LIN {X 0,Y 566.227,Z 211.515,A -85,B 0,C 180,E1 -2635.049,E2 -2635.049} C_VEL
LIN {X 0,Y 566.206,Z 211.459,A -85,B 0,C 180,E1 -2638.202,E2 -2638.202} C_VEL
LIN {X 0,Y 566.191,Z 211.454,A -85,B 0,C 180,E1 -2641.076,E2 -2641.076} C_VEL
LIN {X 0,Y 566.214,Z 211.456,A -85,B 0,C 180,E1 -2643.734,E2 -2643.734} C_VEL
LIN {X 0,Y 566.201,Z 211.452,A -85,B 0,C 180,E1 -2646.57,E2 -2646.57} C_VEL
LIN {X 0,Y 566.223,Z 211.456,A -85,B 0,C 180,E1 -2649.686,E2 -2649.686} C_VEL
LIN {X 0,Y 566.202,Z 211.451,A -85,B 0,C 180,E1 -2652.917,E2 -2652.917} C_VEL
LIN {X 0,Y 566.199,Z 211.455,A -85,B 0,C 180,E1 -2656.048,E2 -2656.048} C_VEL
LIN {X 0,Y 566.205,Z 211.454,A -85,B 0,C 180,E1 -2659.214,E2 -2659.214} C_VEL
LIN {X 0,Y 566.186,Z 211.462,A -85,B 0,C 180,E1 -2661.636,E2 -2661.636} C_VEL
LIN {X 0,Y 566.162,Z 211.455,A -85,B 0,C 180,E1 -2664.307,E2 -2664.307} C_VEL
LIN {X 0,Y 566.204,Z 211.45,A -85,B 0,C 180,E1 -2666.896,E2 -2666.896} C_VEL
LIN {X 0,Y 566.176,Z 211.464,A -85,B 0,C 180,E1 -2669.407,E2 -2669.407} C_VEL
LIN {X 0,Y 566.212,Z 211.45,A -85,B 0,C 180,E1 -2671.857,E2 -2671.857} C_VEL
LIN {X 0,Y 566.21,Z 211.448,A -85,B 0,C 180,E1 -2674.25,E2 -2674.25} C_VEL
LIN {X 0,Y 566.172,Z 211.456,A -85,B 0,C 180,E1 -2676.718,E2 -2676.718} C_VEL
LIN {X 0,Y 566.207,Z 211.45,A -85,B 0,C 180,E1 -2679.662,E2 -2679.662} C_VEL
LIN {X 0,Y 566.197,Z 211.45,A -85,B 0,C 180,E1 -2682.668,E2 -2682.668} C_VEL
LIN {X 0,Y 566.234,Z 211.449,A -85,B 0,C 180,E1 -2685.626,E2 -2685.626} C_VEL
LIN {X 0,Y 566.235,Z 211.449,A -85,B 0,C 180,E1 -2688.675,E2 -2688.675} C_VEL
LIN {X 0,Y 566.206,Z 211.451,A -85,B 0,C 180,E1 -2691.434,E2 -2691.434} C_VEL
LIN {X 0,Y 566.264,Z 211.444,A -85,B 0,C 180,E1 -2694.301,E2 -2694.301} C_VEL
LIN {X 0,Y 566.283,Z 211.439,A -85,B 0,C 180,E1 -2697.866,E2 -2697.866} C_VEL
LIN {X 0,Y 566.305,Z 211.441,A -85,B 0,C 180,E1 -2700.711,E2 -2700.711} C_VEL
LIN {X 0,Y 566.271,Z 211.45,A -85,B 0,C 180,E1 -2702.845,E2 -2702.845} C_VEL
LIN {X 0,Y 566.262,Z 211.443,A -85,B 0,C 180,E1 -2705.698,E2 -2705.698} C_VEL
LIN {X 0,Y 566.233,Z 211.454,A -85,B 0,C 180,E1 -2708.565,E2 -2708.565} C_VEL
LIN {X 0,Y 566.24,Z 211.444,A -85,B 0,C 180,E1 -2711.454,E2 -2711.454} C_VEL
LIN {X 0,Y 566.233,Z 211.457,A -85,B 0,C 180,E1 -2714.506,E2 -2714.506} C_VEL
LIN {X 0,Y 566.198,Z 211.45,A -85,B 0,C 180,E1 -2717.331,E2 -2717.331} C_VEL
LIN {X 0,Y 566.212,Z 211.454,A -85,B 0,C 180,E1 -2720.337,E2 -2720.337} C_VEL
LIN {X 0,Y 566.167,Z 211.455,A -85,B 0,C 180,E1 -2723.281,E2 -2723.281} C_VEL
LIN {X 0,Y 566.212,Z 211.451,A -85,B 0,C 180,E1 -2725.749,E2 -2725.749} C_VEL
LIN {X 0,Y 566.2,Z 211.448,A -85,B 0,C 180,E1 -2727.484,E2 -2727.484} C_VEL
LIN {X 0,Y 565.52,Z 211.54,A -85,B 0,C 180,E1 -2728.078,E2 -2728.078} C_VEL
LIN {X 0,Y 562.655,Z 211.899,A -85,B 0,C 180,E1 -2729.042,E2 -2729.042} C_VEL
LIN {X 0,Y 560.247,Z 212.2,A -85,B 0,C 180,E1 -2729.817,E2 -2729.817} C_VEL
LIN {X 0,Y 559.221,Z 212.327,A -85,B 0,C 180,E1 -2730.416,E2 -2730.416} C_VEL
LIN {X 0,Y 559.142,Z 212.333,A -85,B 0,C 180,E1 -2730.619,E2 -2730.619} C_VEL
LIN {X 0,Y 559.162,Z 212.329,A -85,B 0,C 180,E1 -2733.574,E2 -2733.574} C_VEL
LIN {X 0,Y 559.159,Z 212.333,A -85,B 0,C 180,E1 -2736.447,E2 -2736.447} C_VEL
LIN {X 0,Y 559.176,Z 212.326,A -85,B 0,C 180,E1 -2738.933,E2 -2738.933} C_VEL
LIN {X 0,Y 559.189,Z 212.329,A -85,B 0,C 180,E1 -2741.767,E2 -2741.767} C_VEL
LIN {X 0,Y 559.137,Z 212.33,A -85,B 0,C 180,E1 -2744.739,E2 -2744.739} C_VEL
LIN {X 0,Y 559.174,Z 212.327,A -85,B 0,C 180,E1 -2747.862,E2 -2747.862} C_VEL
LIN {X 0,Y 559.182,Z 212.33,A -85,B 0,C 180,E1 -2750.135,E2 -2750.135} C_VEL
LIN {X 0,Y 559.141,Z 212.331,A -85,B 0,C 180,E1 -2752.892,E2 -2752.892} C_VEL
LIN {X 0,Y 559.162,Z 212.331,A -85,B 0,C 180,E1 -2756.051,E2 -2756.051} C_VEL
LIN {X 0,Y 559.16,Z 212.33,A -85,B 0,C 180,E1 -2758.981,E2 -2758.981} C_VEL
LIN {X 0,Y 559.189,Z 212.326,A -85,B 0,C 180,E1 -2762.288,E2 -2762.288} C_VEL
LIN {X 0,Y 559.176,Z 212.328,A -85,B 0,C 180,E1 -2764.813,E2 -2764.813} C_VEL
LIN {X 0,Y 559.139,Z 212.335,A -85,B 0,C 180,E1 -2767.847,E2 -2767.847} C_VEL
LIN {X 0,Y 559.194,Z 212.325,A -85,B 0,C 180,E1 -2770.492,E2 -2770.492} C_VEL
LIN {X 0,Y 559.178,Z 212.335,A -85,B 0,C 180,E1 -2773.198,E2 -2773.198} C_VEL
LIN {X 0,Y 559.169,Z 212.328,A -85,B 0,C 180,E1 -2776.184,E2 -2776.184} C_VEL
LIN {X 0,Y 559.194,Z 212.333,A -85,B 0,C 180,E1 -2779.134,E2 -2779.134} C_VEL
LIN {X 0,Y 559.203,Z 212.324,A -85,B 0,C 180,E1 -2782.054,E2 -2782.054} C_VEL
LIN {X 0,Y 559.253,Z 212.325,A -85,B 0,C 180,E1 -2784.953,E2 -2784.953} C_VEL
LIN {X 0,Y 559.255,Z 212.318,A -85,B 0,C 180,E1 -2787.839,E2 -2787.839} C_VEL
LIN {X 0,Y 559.27,Z 212.322,A -85,B 0,C 180,E1 -2790.72,E2 -2790.72} C_VEL
LIN {X 0,Y 559.236,Z 212.328,A -85,B 0,C 180,E1 -2792.881,E2 -2792.881} C_VEL
LIN {X 0,Y 559.236,Z 212.32,A -85,B 0,C 180,E1 -2795.77,E2 -2795.77} C_VEL
LIN {X 0,Y 559.189,Z 212.333,A -85,B 0,C 180,E1 -2798.674,E2 -2798.674} C_VEL
LIN {X 0,Y 559.202,Z 212.325,A -85,B 0,C 180,E1 -2801.6,E2 -2801.6} C_VEL
LIN {X 0,Y 559.197,Z 212.333,A -85,B 0,C 180,E1 -2804.596,E2 -2804.596} C_VEL
LIN {X 0,Y 559.156,Z 212.33,A -85,B 0,C 180,E1 -2807.557,E2 -2807.557} C_VEL
LIN {X 0,Y 559.169,Z 212.329,A -85,B 0,C 180,E1 -2809.837,E2 -2809.837} C_VEL
LIN {X 0,Y 559.139,Z 212.335,A -85,B 0,C 180,E1 -2812.153,E2 -2812.153} C_VEL
LIN {X 0,Y 559.173,Z 212.328,A -85,B 0,C 180,E1 -2815.298,E2 -2815.298} C_VEL
LIN {X 0,Y 559.189,Z 212.326,A -85,B 0,C 180,E1 -2817.712,E2 -2817.712} C_VEL
LIN {X 0,Y 559.16,Z 212.33,A -85,B 0,C 180,E1 -2821.019,E2 -2821.019} C_VEL
LIN {X 0,Y 559.162,Z 212.331,A -85,B 0,C 180,E1 -2823.949,E2 -2823.949} C_VEL
LIN {X 0,Y 559.141,Z 212.331,A -85,B 0,C 180,E1 -2827.108,E2 -2827.108} C_VEL
LIN {X 0,Y 559.167,Z 212.333,A -85,B 0,C 180,E1 -2829.943,E2 -2829.943} C_VEL
LIN {X 0,Y 559.161,Z 212.324,A -85,B 0,C 180,E1 -2832.743,E2 -2832.743} C_VEL
LIN {X 0,Y 559.152,Z 212.333,A -85,B 0,C 180,E1 -2835.761,E2 -2835.761} C_VEL
LIN {X 0,Y 559.189,Z 212.329,A -85,B 0,C 180,E1 -2838.233,E2 -2838.233} C_VEL
LIN {X 0,Y 559.175,Z 212.327,A -85,B 0,C 180,E1 -2841.191,E2 -2841.191} C_VEL
LIN {X 0,Y 559.158,Z 212.336,A -85,B 0,C 180,E1 -2843.791,E2 -2843.791} C_VEL
LIN {X 0,Y 559.162,Z 212.329,A -85,B 0,C 180,E1 -2846.426,E2 -2846.426} C_VEL
LIN {X 0,Y 559.16,Z 212.329,A -85,B 0,C 180,E1 -2848.982,E2 -2848.982} C_VEL
LIN {X 0,Y 559.165,Z 212.334,A -85,B 0,C 180,E1 -2851.619,E2 -2851.619} C_VEL
LIN {X 0,Y 559.179,Z 212.332,A -85,B 0,C 180,E1 -2853.903,E2 -2853.903} C_VEL
LIN {X 0,Y 559.14,Z 212.331,A -85,B 0,C 180,E1 -2856.571,E2 -2856.571} C_VEL
LIN {X 0,Y 559.178,Z 212.331,A -85,B 0,C 180,E1 -2859.396,E2 -2859.396} C_VEL
LIN {X 0,Y 559.145,Z 212.336,A -85,B 0,C 180,E1 -2861.686,E2 -2861.686} C_VEL
LIN {X 0,Y 559.165,Z 212.331,A -85,B 0,C 180,E1 -2863.948,E2 -2863.948} C_VEL
LIN {X 0,Y 559.17,Z 212.328,A -85,B 0,C 180,E1 -2866.184,E2 -2866.184} C_VEL
LIN {X 0,Y 559.195,Z 212.326,A -85,B 0,C 180,E1 -2869.134,E2 -2869.134} C_VEL
LIN {X 0,Y 559.201,Z 212.322,A -85,B 0,C 180,E1 -2872.054,E2 -2872.054} C_VEL
LIN {X 0,Y 559.254,Z 212.321,A -85,B 0,C 180,E1 -2874.954,E2 -2874.954} C_VEL
LIN {X 0,Y 559.256,Z 212.315,A -85,B 0,C 180,E1 -2877.84,E2 -2877.84} C_VEL
LIN {X 0,Y 559.268,Z 212.312,A -85,B 0,C 180,E1 -2880.72,E2 -2880.72} C_VEL
LIN {X 0,Y 559.234,Z 212.323,A -85,B 0,C 180,E1 -2882.882,E2 -2882.882} C_VEL
LIN {X 0,Y 559.231,Z 212.32,A -85,B 0,C 180,E1 -2885.771,E2 -2885.771} C_VEL
LIN {X 0,Y 559.17,Z 212.328,A -85,B 0,C 180,E1 -2888.675,E2 -2888.675} C_VEL
LIN {X 0,Y 559.205,Z 212.322,A -85,B 0,C 180,E1 -2891.601,E2 -2891.601} C_VEL
LIN {X 0,Y 559.2,Z 212.328,A -85,B 0,C 180,E1 -2894.596,E2 -2894.596} C_VEL
LIN {X 0,Y 559.14,Z 212.327,A -85,B 0,C 180,E1 -2897.558,E2 -2897.558} C_VEL
LIN {X 0,Y 559.166,Z 212.324,A -85,B 0,C 180,E1 -2899.838,E2 -2899.838} C_VEL
LIN {X 0,Y 559.141,Z 212.331,A -85,B 0,C 180,E1 -2902.153,E2 -2902.153} C_VEL
LIN {X 0,Y 559.176,Z 212.325,A -85,B 0,C 180,E1 -2905.299,E2 -2905.299} C_VEL
LIN {X 0,Y 559.157,Z 212.325,A -85,B 0,C 180,E1 -2907.714,E2 -2907.714} C_VEL
LIN {X 0,Y 559.15,Z 212.333,A -85,B 0,C 180,E1 -2910.183,E2 -2910.183} C_VEL
LIN {X 0,Y 559.153,Z 212.333,A -85,B 0,C 180,E1 -2912.716,E2 -2912.716} C_VEL
LIN {X 0,Y 559.128,Z 212.331,A -85,B 0,C 180,E1 -2915.324,E2 -2915.324} C_VEL
LIN {X 0,Y 559.133,Z 212.335,A -85,B 0,C 180,E1 -2918.018,E2 -2918.018} C_VEL
LIN {X 0,Y 559.156,Z 212.332,A -85,B 0,C 180,E1 -2920.813,E2 -2920.813} C_VEL
LIN {X 0,Y 559.142,Z 212.332,A -85,B 0,C 180,E1 -2923.734,E2 -2923.734} C_VEL
LIN {X 0,Y 559.146,Z 212.332,A -85,B 0,C 180,E1 -2926.804,E2 -2926.804} C_VEL
LIN {X 0,Y 559.157,Z 212.325,A -85,B 0,C 180,E1 -2929.188,E2 -2929.188} C_VEL
LIN {X 0,Y 559.134,Z 212.338,A -85,B 0,C 180,E1 -2931.983,E2 -2931.983} C_VEL
LIN {X 0,Y 559.132,Z 212.332,A -85,B 0,C 180,E1 -2934.788,E2 -2934.788} C_VEL
LIN {X 0,Y 559.157,Z 212.33,A -85,B 0,C 180,E1 -2937.365,E2 -2937.365} C_VEL
LIN {X 0,Y 559.149,Z 212.337,A -85,B 0,C 180,E1 -2940.143,E2 -2940.143} C_VEL
LIN {X 0,Y 559.162,Z 212.332,A -85,B 0,C 180,E1 -2943.175,E2 -2943.175} C_VEL
LIN {X 0,Y 559.193,Z 212.546,A -85,B 0,C 180,E1 -2944.845,E2 -2944.845} C_VEL
LIN {X 0,Y 559.929,Z 217.985,A -85,B 0,C 180,E1 -2945.925,E2 -2945.925} C_VEL
LIN {X 0,Y 559.641,Z 232.53,A -85,B 0,C 180,E1 -2948.643,E2 -2948.643} C_VEL
LIN {X 0,Y 559.484,Z 246.129,A -85,B 0,C 180,E1 -2951.128,E2 -2951.128} C_VEL
LIN {X 0,Y 559.339,Z 260.753,A -85,B 0,C 180,E1 -2953.766,E2 -2953.766} C_VEL
LIN {X 0,Y 559.262,Z 272.268,A -85,B 0,C 180,E1 -2955.792,E2 -2955.792} C_VEL
LIN {X 0,Y 559.599,Z 274.63,A -85,B 0,C 180,E1 -2955.869,E2 -2955.869} C_VEL
LIN {X 0,Y 560.277,Z 280.09,A -85,B 0,C 180,E1 -2955.957,E2 -2955.957} C_VEL
LIN {X 0,Y 560.031,Z 378.524,A -85,B 0,C 180,E1 -2957.245,E2 -2957.245} C_VEL
LIN {X 0,Y 559.963,Z 388.812,A -85,B 0,C 180,E1 -2957.473,E2 -2957.473} C_VEL
LIN {X 0,Y 559.826,Z 399.596,A -85,B 0,C 180,E1 -2957.816,E2 -2957.816} C_VEL
LIN {X 0,Y 559.716,Z 412.055,A -85,B 0,C 180,E1 -2958.351,E2 -2958.351} C_VEL
LIN {X 0,Y 559.537,Z 424.284,A -85,B 0,C 180,E1 -2959.06,E2 -2959.06} C_VEL
LIN {X 0,Y 559.434,Z 433.031,A -85,B 0,C 180,E1 -2959.687,E2 -2959.687} C_VEL
LIN {X 0,Y 559.277,Z 441.533,A -85,B 0,C 180,E1 -2960.416,E2 -2960.416} C_VEL
LIN {X 0,Y 559.138,Z 448.723,A -85,B 0,C 180,E1 -2961.143,E2 -2961.143} C_VEL
LIN {X 0,Y 559.052,Z 456.27,A -85,B 0,C 180,E1 -2962.051,E2 -2962.051} C_VEL
LIN {X 0,Y 558.934,Z 462.674,A -85,B 0,C 180,E1 -2962.976,E2 -2962.976} C_VEL
LIN {X 0,Y 558.909,Z 467.794,A -85,B 0,C 180,E1 -2963.864,E2 -2963.864} C_VEL
LIN {X 0,Y 558.798,Z 472.891,A -85,B 0,C 180,E1 -2964.949,E2 -2964.949} C_VEL
LIN {X 0,Y 558.844,Z 476.848,A -85,B 0,C 180,E1 -2966.034,E2 -2966.034} C_VEL
LIN {X 0,Y 558.799,Z 479.771,A -85,B 0,C 180,E1 -2967.116,E2 -2967.116} C_VEL
LIN {X 0,Y 558.745,Z 482.196,A -85,B 0,C 180,E1 -2968.559,E2 -2968.559} C_VEL
LIN {X 0,Y 558.741,Z 482.78,A -85,B 0,C 180,E1 -2969.279,E2 -2969.279} C_VEL
LIN {X 0,Y 558.741,Z 482.78,A -85,B 0,C 180,E1 -2970.721,E2 -2970.721} C_VEL
LIN {X 0,Y 558.745,Z 482.196,A -85,B 0,C 180,E1 -2971.441,E2 -2971.441} C_VEL
LIN {X 0,Y 558.799,Z 479.771,A -85,B 0,C 180,E1 -2972.884,E2 -2972.884} C_VEL
LIN {X 0,Y 558.844,Z 476.848,A -85,B 0,C 180,E1 -2973.966,E2 -2973.966} C_VEL
LIN {X 0,Y 558.798,Z 472.891,A -85,B 0,C 180,E1 -2975.051,E2 -2975.051} C_VEL
LIN {X 0,Y 558.91,Z 467.794,A -85,B 0,C 180,E1 -2976.136,E2 -2976.136} C_VEL
LIN {X 0,Y 558.934,Z 462.674,A -85,B 0,C 180,E1 -2977.024,E2 -2977.024} C_VEL
LIN {X 0,Y 559.052,Z 456.27,A -85,B 0,C 180,E1 -2977.949,E2 -2977.949} C_VEL
LIN {X 0,Y 559.138,Z 448.723,A -85,B 0,C 180,E1 -2978.857,E2 -2978.857} C_VEL
LIN {X 0,Y 559.287,Z 439.616,A -85,B 0,C 180,E1 -2979.767,E2 -2979.767} C_VEL
LIN {X 0,Y 559.46,Z 428.158,A -85,B 0,C 180,E1 -2980.678,E2 -2980.678} C_VEL
LIN {X 0,Y 559.566,Z 419.19,A -85,B 0,C 180,E1 -2981.257,E2 -2981.257} C_VEL
LIN {X 0,Y 559.75,Z 408.68,A -85,B 0,C 180,E1 -2981.805,E2 -2981.805} C_VEL
LIN {X 0,Y 559.826,Z 399.596,A -85,B 0,C 180,E1 -2982.184,E2 -2982.184} C_VEL
LIN {X 0,Y 559.963,Z 388.812,A -85,B 0,C 180,E1 -2982.527,E2 -2982.527} C_VEL
LIN {X 0,Y 560.031,Z 378.524,A -85,B 0,C 180,E1 -2982.755,E2 -2982.755} C_VEL
LIN {X 0,Y 560.215,Z 278.301,A -85,B 0,C 180,E1 -2984.067,E2 -2984.067} C_VEL
LIN {X 0,Y 559.276,Z 272.599,A -85,B 0,C 180,E1 -2984.184,E2 -2984.184} C_VEL
LIN {X 0,Y 559.225,Z 271.167,A -85,B 0,C 180,E1 -2984.371,E2 -2984.371} C_VEL
LIN {X 0,Y 559.399,Z 254.896,A -85,B 0,C 180,E1 -2987.287,E2 -2987.287} C_VEL
LIN {X 0,Y 559.617,Z 238.81,A -85,B 0,C 180,E1 -2990.204,E2 -2990.204} C_VEL
LIN {X 0,Y 559.874,Z 222.392,A -85,B 0,C 180,E1 -2993.25,E2 -2993.25} C_VEL
LIN {X 0,Y 559.783,Z 215.926,A -85,B 0,C 180,E1 -2994.476,E2 -2994.476} C_VEL
LIN {X 0,Y 559.186,Z 212.411,A -85,B 0,C 180,E1 -2995.188,E2 -2995.188} C_VEL
LIN {X 0,Y 559.139,Z 212.339,A -85,B 0,C 180,E1 -2997.714,E2 -2997.714} C_VEL
LIN {X 0,Y 559.154,Z 212.338,A -85,B 0,C 180,E1 -3000.183,E2 -3000.183} C_VEL
LIN {X 0,Y 559.158,Z 212.329,A -85,B 0,C 180,E1 -3002.715,E2 -3002.715} C_VEL
LIN {X 0,Y 559.129,Z 212.334,A -85,B 0,C 180,E1 -3005.324,E2 -3005.324} C_VEL
LIN {X 0,Y 559.135,Z 212.338,A -85,B 0,C 180,E1 -3008.017,E2 -3008.017} C_VEL
LIN {X 0,Y 559.157,Z 212.325,A -85,B 0,C 180,E1 -3010.812,E2 -3010.812} C_VEL
LIN {X 0,Y 559.157,Z 212.338,A -85,B 0,C 180,E1 -3013.732,E2 -3013.732} C_VEL
LIN {X 0,Y 559.148,Z 212.33,A -85,B 0,C 180,E1 -3016.803,E2 -3016.803} C_VEL
LIN {X 0,Y 559.156,Z 212.332,A -85,B 0,C 180,E1 -3019.187,E2 -3019.187} C_VEL
LIN {X 0,Y 559.133,Z 212.335,A -85,B 0,C 180,E1 -3021.982,E2 -3021.982} C_VEL
LIN {X 0,Y 559.131,Z 212.331,A -85,B 0,C 180,E1 -3024.787,E2 -3024.787} C_VEL
LIN {X 0,Y 559.154,Z 212.335,A -85,B 0,C 180,E1 -3027.364,E2 -3027.364} C_VEL
LIN {X 0,Y 559.145,Z 212.33,A -85,B 0,C 180,E1 -3030.143,E2 -3030.143} C_VEL
LIN {X 0,Y 559.17,Z 212.33,A -85,B 0,C 180,E1 -3033.097,E2 -3033.097} C_VEL
LIN {X 0,Y 559.156,Z 212.335,A -85,B 0,C 180,E1 -3035.494,E2 -3035.494} C_VEL
LIN {X 0,Y 559.172,Z 212.328,A -85,B 0,C 180,E1 -3038.623,E2 -3038.623} C_VEL
LIN {X 0,Y 559.161,Z 212.33,A -85,B 0,C 180,E1 -3040.926,E2 -3040.926} C_VEL
LIN {X 0,Y 559.163,Z 212.327,A -85,B 0,C 180,E1 -3043.947,E2 -3043.947} C_VEL
LIN {X 0,Y 559.17,Z 212.327,A -85,B 0,C 180,E1 -3046.184,E2 -3046.184} C_VEL
LIN {X 0,Y 559.194,Z 212.326,A -85,B 0,C 180,E1 -3049.133,E2 -3049.133} C_VEL
LIN {X 0,Y 559.196,Z 212.321,A -85,B 0,C 180,E1 -3052.053,E2 -3052.053} C_VEL
LIN {X 0,Y 559.251,Z 212.326,A -85,B 0,C 180,E1 -3054.953,E2 -3054.953} C_VEL
LIN {X 0,Y 559.254,Z 212.315,A -85,B 0,C 180,E1 -3057.839,E2 -3057.839} C_VEL
LIN {X 0,Y 559.274,Z 212.316,A -85,B 0,C 180,E1 -3060.72,E2 -3060.72} C_VEL
LIN {X 0,Y 559.237,Z 212.326,A -85,B 0,C 180,E1 -3062.881,E2 -3062.881} C_VEL
LIN {X 0,Y 559.231,Z 212.319,A -85,B 0,C 180,E1 -3065.77,E2 -3065.77} C_VEL
LIN {X 0,Y 559.191,Z 212.328,A -85,B 0,C 180,E1 -3068.674,E2 -3068.674} C_VEL
LIN {X 0,Y 559.204,Z 212.32,A -85,B 0,C 180,E1 -3071.6,E2 -3071.6} C_VEL
LIN {X 0,Y 559.198,Z 212.332,A -85,B 0,C 180,E1 -3074.595,E2 -3074.595} C_VEL
LIN {X 0,Y 559.157,Z 212.326,A -85,B 0,C 180,E1 -3077.557,E2 -3077.557} C_VEL
LIN {X 0,Y 559.17,Z 212.324,A -85,B 0,C 180,E1 -3079.837,E2 -3079.837} C_VEL
LIN {X 0,Y 559.139,Z 212.336,A -85,B 0,C 180,E1 -3082.152,E2 -3082.152} C_VEL
LIN {X 0,Y 559.174,Z 212.325,A -85,B 0,C 180,E1 -3085.298,E2 -3085.298} C_VEL
LIN {X 0,Y 559.154,Z 212.326,A -85,B 0,C 180,E1 -3087.713,E2 -3087.713} C_VEL
LIN {X 0,Y 559.142,Z 212.333,A -85,B 0,C 180,E1 -3090.619,E2 -3090.619} C_VEL
LIN {X 0,Y 558.483,Z 212.415,A -85,B 0,C 180,E1 -3091.22,E2 -3091.22} C_VEL
LIN {X 0,Y 555.622,Z 212.777,A -85,B 0,C 180,E1 -3092.196,E2 -3092.196} C_VEL
LIN {X 0,Y 553.208,Z 213.072,A -85,B 0,C 180,E1 -3092.982,E2 -3092.982} C_VEL
LIN {X 0,Y 552.185,Z 213.198,A -85,B 0,C 180,E1 -3093.589,E2 -3093.589} C_VEL
LIN {X 0,Y 552.11,Z 213.209,A -85,B 0,C 180,E1 -3093.794,E2 -3093.794} C_VEL
LIN {X 0,Y 552.107,Z 213.208,A -85,B 0,C 180,E1 -3096.746,E2 -3096.746} C_VEL
LIN {X 0,Y 552.131,Z 213.206,A -85,B 0,C 180,E1 -3099.526,E2 -3099.526} C_VEL
LIN {X 0,Y 552.128,Z 213.207,A -85,B 0,C 180,E1 -3102.425,E2 -3102.425} C_VEL
LIN {X 0,Y 552.096,Z 213.212,A -85,B 0,C 180,E1 -3105.563,E2 -3105.563} C_VEL
LIN {X 0,Y 552.137,Z 213.197,A -85,B 0,C 180,E1 -3108.676,E2 -3108.676} C_VEL
LIN {X 0,Y 552.117,Z 213.209,A -85,B 0,C 180,E1 -3111.411,E2 -3111.411} C_VEL
LIN {X 0,Y 552.098,Z 213.207,A -85,B 0,C 180,E1 -3114.157,E2 -3114.157} C_VEL
LIN {X 0,Y 552.12,Z 213.204,A -85,B 0,C 180,E1 -3116.815,E2 -3116.815} C_VEL
LIN {X 0,Y 552.104,Z 213.214,A -85,B 0,C 180,E1 -3119.391,E2 -3119.391} C_VEL
LIN {X 0,Y 552.123,Z 213.21,A -85,B 0,C 180,E1 -3121.903,E2 -3121.903} C_VEL
LIN {X 0,Y 552.152,Z 213.202,A -85,B 0,C 180,E1 -3124.649,E2 -3124.649} C_VEL
LIN {X 0,Y 552.09,Z 213.218,A -85,B 0,C 180,E1 -3127.549,E2 -3127.549} C_VEL
LIN {X 0,Y 552.145,Z 213.203,A -85,B 0,C 180,E1 -3130.373,E2 -3130.373} C_VEL
LIN {X 0,Y 552.152,Z 213.207,A -85,B 0,C 180,E1 -3132.977,E2 -3132.977} C_VEL
LIN {X 0,Y 552.133,Z 213.206,A -85,B 0,C 180,E1 -3136.004,E2 -3136.004} C_VEL
LIN {X 0,Y 552.161,Z 213.208,A -85,B 0,C 180,E1 -3138.993,E2 -3138.993} C_VEL
LIN {X 0,Y 552.157,Z 213.203,A -85,B 0,C 180,E1 -3141.952,E2 -3141.952} C_VEL
LIN {X 0,Y 552.228,Z 213.199,A -85,B 0,C 180,E1 -3144.889,E2 -3144.889} C_VEL
LIN {X 0,Y 552.225,Z 213.194,A -85,B 0,C 180,E1 -3147.812,E2 -3147.812} C_VEL
LIN {X 0,Y 552.24,Z 213.198,A -85,B 0,C 180,E1 -3150.729,E2 -3150.729} C_VEL
LIN {X 0,Y 552.202,Z 213.204,A -85,B 0,C 180,E1 -3152.918,E2 -3152.918} C_VEL
LIN {X 0,Y 552.207,Z 213.196,A -85,B 0,C 180,E1 -3155.844,E2 -3155.844} C_VEL
LIN {X 0,Y 552.159,Z 213.21,A -85,B 0,C 180,E1 -3158.786,E2 -3158.786} C_VEL
LIN {X 0,Y 552.16,Z 213.202,A -85,B 0,C 180,E1 -3161.75,E2 -3161.75} C_VEL
LIN {X 0,Y 552.134,Z 213.213,A -85,B 0,C 180,E1 -3164.748,E2 -3164.748} C_VEL
LIN {X 0,Y 552.108,Z 213.208,A -85,B 0,C 180,E1 -3167.788,E2 -3167.788} C_VEL
LIN {X 0,Y 552.128,Z 213.208,A -85,B 0,C 180,E1 -3170.101,E2 -3170.101} C_VEL
LIN {X 0,Y 552.09,Z 213.218,A -85,B 0,C 180,E1 -3172.451,E2 -3172.451} C_VEL
LIN {X 0,Y 552.152,Z 213.202,A -85,B 0,C 180,E1 -3175.351,E2 -3175.351} C_VEL
LIN {X 0,Y 552.123,Z 213.21,A -85,B 0,C 180,E1 -3178.097,E2 -3178.097} C_VEL
LIN {X 0,Y 552.104,Z 213.214,A -85,B 0,C 180,E1 -3180.609,E2 -3180.609} C_VEL
LIN {X 0,Y 552.12,Z 213.204,A -85,B 0,C 180,E1 -3183.185,E2 -3183.185} C_VEL
LIN {X 0,Y 552.098,Z 213.207,A -85,B 0,C 180,E1 -3185.843,E2 -3185.843} C_VEL
LIN {X 0,Y 552.123,Z 213.205,A -85,B 0,C 180,E1 -3189.062,E2 -3189.062} C_VEL
LIN {X 0,Y 552.137,Z 213.198,A -85,B 0,C 180,E1 -3191.444,E2 -3191.444} C_VEL
LIN {X 0,Y 552.093,Z 213.211,A -85,B 0,C 180,E1 -3194.532,E2 -3194.532} C_VEL
LIN {X 0,Y 552.128,Z 213.207,A -85,B 0,C 180,E1 -3197.585,E2 -3197.585} C_VEL
LIN {X 0,Y 552.132,Z 213.206,A -85,B 0,C 180,E1 -3200.474,E2 -3200.474} C_VEL
LIN {X 0,Y 552.109,Z 213.208,A -85,B 0,C 180,E1 -3203.316,E2 -3203.316} C_VEL
LIN {X 0,Y 552.125,Z 213.211,A -85,B 0,C 180,E1 -3205.94,E2 -3205.94} C_VEL
LIN {X 0,Y 552.116,Z 213.207,A -85,B 0,C 180,E1 -3208.541,E2 -3208.541} C_VEL
LIN {X 0,Y 552.122,Z 213.208,A -85,B 0,C 180,E1 -3211.438,E2 -3211.438} C_VEL
LIN {X 0,Y 552.128,Z 213.204,A -85,B 0,C 180,E1 -3214.356,E2 -3214.356} C_VEL
LIN {X 0,Y 552.097,Z 213.208,A -85,B 0,C 180,E1 -3216.758,E2 -3216.758} C_VEL
LIN {X 0,Y 552.119,Z 213.207,A -85,B 0,C 180,E1 -3219.12,E2 -3219.12} C_VEL
LIN {X 0,Y 552.124,Z 213.206,A -85,B 0,C 180,E1 -3221.445,E2 -3221.445} C_VEL
LIN {X 0,Y 552.115,Z 213.212,A -85,B 0,C 180,E1 -3223.738,E2 -3223.738} C_VEL
LIN {X 0,Y 552.134,Z 213.205,A -85,B 0,C 180,E1 -3226.005,E2 -3226.005} C_VEL
LIN {X 0,Y 552.162,Z 213.2,A -85,B 0,C 180,E1 -3228.994,E2 -3228.994} C_VEL
LIN {X 0,Y 552.156,Z 213.2,A -85,B 0,C 180,E1 -3231.952,E2 -3231.952} C_VEL
LIN {X 0,Y 552.229,Z 213.195,A -85,B 0,C 180,E1 -3234.889,E2 -3234.889} C_VEL
LIN {X 0,Y 552.227,Z 213.19,A -85,B 0,C 180,E1 -3237.812,E2 -3237.812} C_VEL
LIN {X 0,Y 552.238,Z 213.187,A -85,B 0,C 180,E1 -3240.73,E2 -3240.73} C_VEL
LIN {X 0,Y 552.202,Z 213.199,A -85,B 0,C 180,E1 -3242.919,E2 -3242.919} C_VEL
LIN {X 0,Y 552.2,Z 213.195,A -85,B 0,C 180,E1 -3245.844,E2 -3245.844} C_VEL
LIN {X 0,Y 552.142,Z 213.205,A -85,B 0,C 180,E1 -3248.786,E2 -3248.786} C_VEL
LIN {X 0,Y 552.163,Z 213.198,A -85,B 0,C 180,E1 -3251.751,E2 -3251.751} C_VEL
LIN {X 0,Y 552.137,Z 213.21,A -85,B 0,C 180,E1 -3254.749,E2 -3254.749} C_VEL
LIN {X 0,Y 552.098,Z 213.203,A -85,B 0,C 180,E1 -3257.789,E2 -3257.789} C_VEL
LIN {X 0,Y 552.126,Z 213.201,A -85,B 0,C 180,E1 -3260.102,E2 -3260.102} C_VEL
LIN {X 0,Y 552.092,Z 213.213,A -85,B 0,C 180,E1 -3262.451,E2 -3262.451} C_VEL
LIN {X 0,Y 552.156,Z 213.199,A -85,B 0,C 180,E1 -3265.351,E2 -3265.351} C_VEL
LIN {X 0,Y 552.11,Z 213.205,A -85,B 0,C 180,E1 -3268.099,E2 -3268.099} C_VEL
LIN {X 0,Y 552.1,Z 213.217,A -85,B 0,C 180,E1 -3270.61,E2 -3270.61} C_VEL
LIN {X 0,Y 552.107,Z 213.205,A -85,B 0,C 180,E1 -3273.187,E2 -3273.187} C_VEL
LIN {X 0,Y 552.086,Z 213.21,A -85,B 0,C 180,E1 -3275.844,E2 -3275.844} C_VEL
LIN {X 0,Y 552.118,Z 213.211,A -85,B 0,C 180,E1 -3278.589,E2 -3278.589} C_VEL
LIN {X 0,Y 552.122,Z 213.205,A -85,B 0,C 180,E1 -3281.446,E2 -3281.446} C_VEL
LIN {X 0,Y 552.094,Z 213.214,A -85,B 0,C 180,E1 -3284.532,E2 -3284.532} C_VEL
LIN {X 0,Y 552.131,Z 213.205,A -85,B 0,C 180,E1 -3287.585,E2 -3287.585} C_VEL
LIN {X 0,Y 552.134,Z 213.208,A -85,B 0,C 180,E1 -3290.473,E2 -3290.473} C_VEL
LIN {X 0,Y 552.108,Z 213.207,A -85,B 0,C 180,E1 -3293.317,E2 -3293.317} C_VEL
LIN {X 0,Y 552.128,Z 213.211,A -85,B 0,C 180,E1 -3295.939,E2 -3295.939} C_VEL
LIN {X 0,Y 552.122,Z 213.209,A -85,B 0,C 180,E1 -3298.541,E2 -3298.541} C_VEL
LIN {X 0,Y 552.107,Z 213.212,A -85,B 0,C 180,E1 -3301.442,E2 -3301.442} C_VEL
LIN {X 0,Y 552.124,Z 213.213,A -85,B 0,C 180,E1 -3304.356,E2 -3304.356} C_VEL
LIN {X 0,Y 552.158,Z 213.415,A -85,B 0,C 180,E1 -3304.685,E2 -3304.685} C_VEL
LIN {X 0,Y 552.99,Z 218.935,A -85,B 0,C 180,E1 -3305.804,E2 -3305.804} C_VEL
LIN {X 0,Y 552.646,Z 234.49,A -85,B 0,C 180,E1 -3308.75,E2 -3308.75} C_VEL
LIN {X 0,Y 552.464,Z 248.087,A -85,B 0,C 180,E1 -3311.264,E2 -3311.264} C_VEL
LIN {X 0,Y 552.308,Z 262.71,A -85,B 0,C 180,E1 -3313.933,E2 -3313.933} C_VEL
LIN {X 0,Y 552.21,Z 272.104,A -85,B 0,C 180,E1 -3315.606,E2 -3315.606} C_VEL
LIN {X 0,Y 552.533,Z 274.407,A -85,B 0,C 180,E1 -3315.684,E2 -3315.684} C_VEL
LIN {X 0,Y 553.381,Z 280.27,A -85,B 0,C 180,E1 -3315.783,E2 -3315.783} C_VEL
LIN {X 0,Y 553.136,Z 377.099,A -85,B 0,C 180,E1 -3317.06,E2 -3317.06} C_VEL
LIN {X 0,Y 553.043,Z 387.872,A -85,B 0,C 180,E1 -3317.291,E2 -3317.291} C_VEL
LIN {X 0,Y 552.932,Z 396.977,A -85,B 0,C 180,E1 -3317.568,E2 -3317.568} C_VEL
LIN {X 0,Y 552.809,Z 406.337,A -85,B 0,C 180,E1 -3317.938,E2 -3317.938} C_VEL
LIN {X 0,Y 552.677,Z 416.63,A -85,B 0,C 180,E1 -3318.456,E2 -3318.456} C_VEL
LIN {X 0,Y 552.528,Z 425.443,A -85,B 0,C 180,E1 -3319.001,E2 -3319.001} C_VEL
LIN {X 0,Y 552.384,Z 434.149,A -85,B 0,C 180,E1 -3319.647,E2 -3319.647} C_VEL
LIN {X 0,Y 552.239,Z 441.521,A -85,B 0,C 180,E1 -3320.292,E2 -3320.292} C_VEL
LIN {X 0,Y 552.122,Z 448.714,A -85,B 0,C 180,E1 -3321.029,E2 -3321.029} C_VEL
LIN {X 0,Y 552.01,Z 454.891,A -85,B 0,C 180,E1 -3321.765,E2 -3321.765} C_VEL
LIN {X 0,Y 551.904,Z 461.399,A -85,B 0,C 180,E1 -3322.684,E2 -3322.684} C_VEL
LIN {X 0,Y 551.808,Z 467.088,A -85,B 0,C 180,E1 -3323.651,E2 -3323.651} C_VEL
LIN {X 0,Y 551.802,Z 471.338,A -85,B 0,C 180,E1 -3324.519,E2 -3324.519} C_VEL
LIN {X 0,Y 551.766,Z 475.632,A -85,B 0,C 180,E1 -3325.617,E2 -3325.617} C_VEL
LIN {X 0,Y 551.75,Z 477.975,A -85,B 0,C 180,E1 -3326.348,E2 -3326.348} C_VEL
LIN {X 0,Y 551.723,Z 479.764,A -85,B 0,C 180,E1 -3327.079,E2 -3327.079} C_VEL
LIN {X 0,Y 551.645,Z 482.191,A -85,B 0,C 180,E1 -3328.54,E2 -3328.54} C_VEL
LIN {X 0,Y 551.641,Z 482.775,A -85,B 0,C 180,E1 -3329.27,E2 -3329.27} C_VEL
LIN {X 0,Y 551.641,Z 482.775,A -85,B 0,C 180,E1 -3330.73,E2 -3330.73} C_VEL
LIN {X 0,Y 551.645,Z 482.191,A -85,B 0,C 180,E1 -3331.46,E2 -3331.46} C_VEL
LIN {X 0,Y 551.723,Z 479.764,A -85,B 0,C 180,E1 -3332.921,E2 -3332.921} C_VEL
LIN {X 0,Y 551.764,Z 476.84,A -85,B 0,C 180,E1 -3334.017,E2 -3334.017} C_VEL
LIN {X 0,Y 551.723,Z 472.882,A -85,B 0,C 180,E1 -3335.116,E2 -3335.116} C_VEL
LIN {X 0,Y 551.837,Z 468.388,A -85,B 0,C 180,E1 -3336.098,E2 -3336.098} C_VEL
LIN {X 0,Y 551.886,Z 462.549,A -85,B 0,C 180,E1 -3337.132,E2 -3337.132} C_VEL
LIN {X 0,Y 551.984,Z 456.261,A -85,B 0,C 180,E1 -3338.051,E2 -3338.051} C_VEL
LIN {X 0,Y 552.071,Z 450.334,A -85,B 0,C 180,E1 -3338.787,E2 -3338.787} C_VEL
LIN {X 0,Y 552.222,Z 443.434,A -85,B 0,C 180,E1 -3339.523,E2 -3339.523} C_VEL
LIN {X 0,Y 552.34,Z 435.28,A -85,B 0,C 180,E1 -3340.261,E2 -3340.261} C_VEL
LIN {X 0,Y 552.479,Z 426.792,A -85,B 0,C 180,E1 -3340.907,E2 -3340.907} C_VEL
LIN {X 0,Y 552.672,Z 417.641,A -85,B 0,C 180,E1 -3341.486,E2 -3341.486} C_VEL
LIN {X 0,Y 552.813,Z 408.352,A -85,B 0,C 180,E1 -3341.969,E2 -3341.969} C_VEL
LIN {X 0,Y 552.9,Z 399.554,A -85,B 0,C 180,E1 -3342.34,E2 -3342.34} C_VEL
LIN {X 0,Y 553.035,Z 389.622,A -85,B 0,C 180,E1 -3342.663,E2 -3342.663} C_VEL
LIN {X 0,Y 553.096,Z 379.762,A -85,B 0,C 180,E1 -3342.895,E2 -3342.895} C_VEL
LIN {X 0,Y 553.264,Z 355.152,A -85,B 0,C 180,E1 -3343.241,E2 -3343.241} C_VEL
LIN {X 0,Y 553.31,Z 278.875,A -85,B 0,C 180,E1 -3344.237,E2 -3344.237} C_VEL
LIN {X 0,Y 552.213,Z 272.296,A -85,B 0,C 180,E1 -3344.379,E2 -3344.379} C_VEL
LIN {X 0,Y 552.313,Z 260.622,A -85,B 0,C 180,E1 -3346.447,E2 -3346.447} C_VEL
LIN {X 0,Y 552.522,Z 245.997,A -85,B 0,C 180,E1 -3349.119,E2 -3349.119} C_VEL
LIN {X 0,Y 552.759,Z 231.34,A -85,B 0,C 180,E1 -3351.851,E2 -3351.851} C_VEL
LIN {X 0,Y 552.979,Z 218.96,A -85,B 0,C 180,E1 -3354.197,E2 -3354.197} C_VEL
LIN {X 0,Y 552.134,Z 213.236,A -85,B 0,C 180,E1 -3355.38,E2 -3355.38} C_VEL
LIN {X 0,Y 552.091,Z 213.217,A -85,B 0,C 180,E1 -3358.099,E2 -3358.099} C_VEL
LIN {X 0,Y 552.103,Z 213.211,A -85,B 0,C 180,E1 -3360.609,E2 -3360.609} C_VEL
LIN {X 0,Y 552.117,Z 213.206,A -85,B 0,C 180,E1 -3363.186,E2 -3363.186} C_VEL
LIN {X 0,Y 552.087,Z 213.215,A -85,B 0,C 180,E1 -3365.843,E2 -3365.843} C_VEL
LIN {X 0,Y 552.126,Z 213.205,A -85,B 0,C 180,E1 -3369.061,E2 -3369.061} C_VEL
LIN {X 0,Y 552.122,Z 213.205,A -85,B 0,C 180,E1 -3371.446,E2 -3371.446} C_VEL
LIN {X 0,Y 552.092,Z 213.209,A -85,B 0,C 180,E1 -3374.531,E2 -3374.531} C_VEL
LIN {X 0,Y 552.131,Z 213.212,A -85,B 0,C 180,E1 -3377.584,E2 -3377.584} C_VEL
LIN {X 0,Y 552.13,Z 213.202,A -85,B 0,C 180,E1 -3380.472,E2 -3380.472} C_VEL
LIN {X 0,Y 552.107,Z 213.213,A -85,B 0,C 180,E1 -3383.317,E2 -3383.317} C_VEL
LIN {X 0,Y 552.103,Z 213.207,A -85,B 0,C 180,E1 -3385.937,E2 -3385.937} C_VEL
LIN {X 0,Y 552.12,Z 213.205,A -85,B 0,C 180,E1 -3388.54,E2 -3388.54} C_VEL
LIN {X 0,Y 552.125,Z 213.21,A -85,B 0,C 180,E1 -3391.438,E2 -3391.438} C_VEL
LIN {X 0,Y 552.129,Z 213.201,A -85,B 0,C 180,E1 -3394.355,E2 -3394.355} C_VEL
LIN {X 0,Y 552.098,Z 213.21,A -85,B 0,C 180,E1 -3396.757,E2 -3396.757} C_VEL
LIN {X 0,Y 552.119,Z 213.213,A -85,B 0,C 180,E1 -3399.119,E2 -3399.119} C_VEL
LIN {X 0,Y 552.118,Z 213.206,A -85,B 0,C 180,E1 -3401.444,E2 -3401.444} C_VEL
LIN {X 0,Y 552.113,Z 213.206,A -85,B 0,C 180,E1 -3403.737,E2 -3403.737} C_VEL
LIN {X 0,Y 552.135,Z 213.203,A -85,B 0,C 180,E1 -3406.004,E2 -3406.004} C_VEL
LIN {X 0,Y 552.162,Z 213.204,A -85,B 0,C 180,E1 -3408.993,E2 -3408.993} C_VEL
LIN {X 0,Y 552.15,Z 213.198,A -85,B 0,C 180,E1 -3411.951,E2 -3411.951} C_VEL
LIN {X 0,Y 552.227,Z 213.201,A -85,B 0,C 180,E1 -3414.889,E2 -3414.889} C_VEL
LIN {X 0,Y 552.225,Z 213.19,A -85,B 0,C 180,E1 -3417.812,E2 -3417.812} C_VEL
LIN {X 0,Y 552.244,Z 213.191,A -85,B 0,C 180,E1 -3420.729,E2 -3420.729} C_VEL
LIN {X 0,Y 552.203,Z 213.201,A -85,B 0,C 180,E1 -3422.918,E2 -3422.918} C_VEL
LIN {X 0,Y 552.201,Z 213.195,A -85,B 0,C 180,E1 -3425.843,E2 -3425.843} C_VEL
LIN {X 0,Y 552.161,Z 213.201,A -85,B 0,C 180,E1 -3428.785,E2 -3428.785} C_VEL
LIN {X 0,Y 552.161,Z 213.197,A -85,B 0,C 180,E1 -3431.75,E2 -3431.75} C_VEL
LIN {X 0,Y 552.135,Z 213.209,A -85,B 0,C 180,E1 -3434.748,E2 -3434.748} C_VEL
LIN {X 0,Y 552.109,Z 213.205,A -85,B 0,C 180,E1 -3437.788,E2 -3437.788} C_VEL
LIN {X 0,Y 552.129,Z 213.203,A -85,B 0,C 180,E1 -3440.101,E2 -3440.101} C_VEL
LIN {X 0,Y 552.09,Z 213.217,A -85,B 0,C 180,E1 -3442.451,E2 -3442.451} C_VEL
LIN {X 0,Y 552.153,Z 213.2,A -85,B 0,C 180,E1 -3445.35,E2 -3445.35} C_VEL
LIN {X 0,Y 552.107,Z 213.209,A -85,B 0,C 180,E1 -3448.098,E2 -3448.098} C_VEL
LIN {X 0,Y 552.104,Z 213.211,A -85,B 0,C 180,E1 -3450.615,E2 -3450.615} C_VEL
LIN {X 0,Y 552.12,Z 213.204,A -85,B 0,C 180,E1 -3453.185,E2 -3453.185} C_VEL
LIN {X 0,Y 552.11,Z 213.209,A -85,B 0,C 180,E1 -3453.794,E2 -3453.794} C_VEL
LIN {X 0,Y 551.473,Z 213.293,A -85,B 0,C 180,E1 -3454.403,E2 -3454.403} C_VEL
LIN {X 0,Y 548.651,Z 213.645,A -85,B 0,C 180,E1 -3455.391,E2 -3455.391} C_VEL
LIN {X 0,Y 546.231,Z 213.947,A -85,B 0,C 180,E1 -3456.186,E2 -3456.186} C_VEL
LIN {X 0,Y 545.163,Z 214.073,A -85,B 0,C 180,E1 -3456.8,E2 -3456.8} C_VEL
LIN {X 0,Y 545.061,Z 214.085,A -85,B 0,C 180,E1 -3457.008,E2 -3457.008} C_VEL
LIN {X 0,Y 545.072,Z 214.087,A -85,B 0,C 180,E1 -3460.141,E2 -3460.141} C_VEL
LIN {X 0,Y 545.083,Z 214.082,A -85,B 0,C 180,E1 -3463.105,E2 -3463.105} C_VEL
LIN {X 0,Y 545.064,Z 214.082,A -85,B 0,C 180,E1 -3466.224,E2 -3466.224} C_VEL
LIN {X 0,Y 545.098,Z 214.073,A -85,B 0,C 180,E1 -3468.887,E2 -3468.887} C_VEL
LIN {X 0,Y 545.052,Z 214.095,A -85,B 0,C 180,E1 -3471.763,E2 -3471.763} C_VEL
LIN {X 0,Y 545.048,Z 214.082,A -85,B 0,C 180,E1 -3474.533,E2 -3474.533} C_VEL
LIN {X 0,Y 545.079,Z 214.084,A -85,B 0,C 180,E1 -3477.212,E2 -3477.212} C_VEL
LIN {X 0,Y 545.063,Z 214.086,A -85,B 0,C 180,E1 -3479.811,E2 -3479.811} C_VEL
LIN {X 0,Y 545.091,Z 214.082,A -85,B 0,C 180,E1 -3482.344,E2 -3482.344} C_VEL
LIN {X 0,Y 545.114,Z 214.08,A -85,B 0,C 180,E1 -3484.82,E2 -3484.82} C_VEL
LIN {X 0,Y 545.035,Z 214.095,A -85,B 0,C 180,E1 -3487.242,E2 -3487.242} C_VEL
LIN {X 0,Y 545.117,Z 214.079,A -85,B 0,C 180,E1 -3490.415,E2 -3490.415} C_VEL
LIN {X 0,Y 545.071,Z 214.091,A -85,B 0,C 180,E1 -3493.521,E2 -3493.521} C_VEL
LIN {X 0,Y 545.092,Z 214.084,A -85,B 0,C 180,E1 -3495.82,E2 -3495.82} C_VEL
LIN {X 0,Y 545.116,Z 214.083,A -85,B 0,C 180,E1 -3498.849,E2 -3498.849} C_VEL
LIN {X 0,Y 545.127,Z 214.079,A -85,B 0,C 180,E1 -3501.847,E2 -3501.847} C_VEL
LIN {X 0,Y 545.205,Z 214.074,A -85,B 0,C 180,E1 -3504.823,E2 -3504.823} C_VEL
LIN {X 0,Y 545.196,Z 214.07,A -85,B 0,C 180,E1 -3507.784,E2 -3507.784} C_VEL
LIN {X 0,Y 545.21,Z 214.074,A -85,B 0,C 180,E1 -3510.739,E2 -3510.739} C_VEL
LIN {X 0,Y 545.169,Z 214.08,A -85,B 0,C 180,E1 -3512.956,E2 -3512.956} C_VEL
LIN {X 0,Y 545.178,Z 214.072,A -85,B 0,C 180,E1 -3515.919,E2 -3515.919} C_VEL
LIN {X 0,Y 545.118,Z 214.087,A -85,B 0,C 180,E1 -3518.9,E2 -3518.9} C_VEL
LIN {X 0,Y 545.132,Z 214.078,A -85,B 0,C 180,E1 -3521.904,E2 -3521.904} C_VEL
LIN {X 0,Y 545.082,Z 214.089,A -85,B 0,C 180,E1 -3524.944,E2 -3524.944} C_VEL
LIN {X 0,Y 545.076,Z 214.086,A -85,B 0,C 180,E1 -3528.026,E2 -3528.026} C_VEL
LIN {X 0,Y 545.092,Z 214.088,A -85,B 0,C 180,E1 -3530.372,E2 -3530.372} C_VEL
LIN {X 0,Y 545.078,Z 214.084,A -85,B 0,C 180,E1 -3533.559,E2 -3533.559} C_VEL
LIN {X 0,Y 545.077,Z 214.086,A -85,B 0,C 180,E1 -3536.001,E2 -3536.001} C_VEL
LIN {X 0,Y 545.087,Z 214.081,A -85,B 0,C 180,E1 -3538.749,E2 -3538.749} C_VEL
LIN {X 0,Y 545.075,Z 214.085,A -85,B 0,C 180,E1 -3541.683,E2 -3541.683} C_VEL
LIN {X 0,Y 545.073,Z 214.084,A -85,B 0,C 180,E1 -3544.564,E2 -3544.564} C_VEL
LIN {X 0,Y 545.037,Z 214.088,A -85,B 0,C 180,E1 -3547.304,E2 -3547.304} C_VEL
LIN {X 0,Y 545.09,Z 214.085,A -85,B 0,C 180,E1 -3550.14,E2 -3550.14} C_VEL
LIN {X 0,Y 545.075,Z 214.076,A -85,B 0,C 180,E1 -3553.107,E2 -3553.107} C_VEL
LIN {X 0,Y 545.061,Z 214.092,A -85,B 0,C 180,E1 -3556.225,E2 -3556.225} C_VEL
LIN {X 0,Y 545.094,Z 214.078,A -85,B 0,C 180,E1 -3558.887,E2 -3558.887} C_VEL
LIN {X 0,Y 545.052,Z 214.092,A -85,B 0,C 180,E1 -3561.763,E2 -3561.763} C_VEL
LIN {X 0,Y 545.05,Z 214.084,A -85,B 0,C 180,E1 -3564.533,E2 -3564.533} C_VEL
LIN {X 0,Y 545.079,Z 214.082,A -85,B 0,C 180,E1 -3567.213,E2 -3567.213} C_VEL
LIN {X 0,Y 545.064,Z 214.093,A -85,B 0,C 180,E1 -3569.811,E2 -3569.811} C_VEL
LIN {X 0,Y 545.078,Z 214.078,A -85,B 0,C 180,E1 -3572.344,E2 -3572.344} C_VEL
LIN {X 0,Y 545.115,Z 214.077,A -85,B 0,C 180,E1 -3574.821,E2 -3574.821} C_VEL
LIN {X 0,Y 545.036,Z 214.091,A -85,B 0,C 180,E1 -3577.243,E2 -3577.243} C_VEL
LIN {X 0,Y 545.119,Z 214.071,A -85,B 0,C 180,E1 -3580.415,E2 -3580.415} C_VEL
LIN {X 0,Y 545.072,Z 214.09,A -85,B 0,C 180,E1 -3583.522,E2 -3583.522} C_VEL
LIN {X 0,Y 545.093,Z 214.085,A -85,B 0,C 180,E1 -3585.82,E2 -3585.82} C_VEL
LIN {X 0,Y 545.117,Z 214.076,A -85,B 0,C 180,E1 -3588.85,E2 -3588.85} C_VEL
LIN {X 0,Y 545.127,Z 214.077,A -85,B 0,C 180,E1 -3591.847,E2 -3591.847} C_VEL
LIN {X 0,Y 545.205,Z 214.069,A -85,B 0,C 180,E1 -3594.823,E2 -3594.823} C_VEL
LIN {X 0,Y 545.198,Z 214.065,A -85,B 0,C 180,E1 -3597.784,E2 -3597.784} C_VEL
LIN {X 0,Y 545.209,Z 214.062,A -85,B 0,C 180,E1 -3600.739,E2 -3600.739} C_VEL
LIN {X 0,Y 545.169,Z 214.076,A -85,B 0,C 180,E1 -3602.956,E2 -3602.956} C_VEL
LIN {X 0,Y 545.17,Z 214.071,A -85,B 0,C 180,E1 -3605.92,E2 -3605.92} C_VEL
LIN {X 0,Y 545.102,Z 214.082,A -85,B 0,C 180,E1 -3608.901,E2 -3608.901} C_VEL
LIN {X 0,Y 545.135,Z 214.073,A -85,B 0,C 180,E1 -3611.905,E2 -3611.905} C_VEL
LIN {X 0,Y 545.086,Z 214.089,A -85,B 0,C 180,E1 -3614.944,E2 -3614.944} C_VEL
LIN {X 0,Y 545.069,Z 214.078,A -85,B 0,C 180,E1 -3618.026,E2 -3618.026} C_VEL
LIN {X 0,Y 545.092,Z 214.08,A -85,B 0,C 180,E1 -3620.373,E2 -3620.373} C_VEL
LIN {X 0,Y 545.08,Z 214.082,A -85,B 0,C 180,E1 -3623.56,E2 -3623.56} C_VEL
LIN {X 0,Y 545.079,Z 214.08,A -85,B 0,C 180,E1 -3626.001,E2 -3626.001} C_VEL
LIN {X 0,Y 545.089,Z 214.088,A -85,B 0,C 180,E1 -3628.748,E2 -3628.748} C_VEL
LIN {X 0,Y 545.055,Z 214.086,A -85,B 0,C 180,E1 -3631.915,E2 -3631.915} C_VEL
LIN {X 0,Y 545.06,Z 214.09,A -85,B 0,C 180,E1 -3634.565,E2 -3634.565} C_VEL
LIN {X 0,Y 545.037,Z 214.088,A -85,B 0,C 180,E1 -3637.304,E2 -3637.304} C_VEL
LIN {X 0,Y 545.066,Z 214.088,A -85,B 0,C 180,E1 -3640.143,E2 -3640.143} C_VEL
LIN {X 0,Y 545.08,Z 214.083,A -85,B 0,C 180,E1 -3643.107,E2 -3643.107} C_VEL
LIN {X 0,Y 545.068,Z 214.093,A -85,B 0,C 180,E1 -3646.225,E2 -3646.225} C_VEL
LIN {X 0,Y 545.083,Z 214.078,A -85,B 0,C 180,E1 -3648.886,E2 -3648.886} C_VEL
LIN {X 0,Y 545.084,Z 214.083,A -85,B 0,C 180,E1 -3650.819,E2 -3650.819} C_VEL
LIN {X 0,Y 545.044,Z 214.089,A -85,B 0,C 180,E1 -3653.62,E2 -3653.62} C_VEL
LIN {X 0,Y 545.067,Z 214.089,A -85,B 0,C 180,E1 -3656.328,E2 -3656.328} C_VEL
LIN {X 0,Y 545.068,Z 214.086,A -85,B 0,C 180,E1 -3658.952,E2 -3658.952} C_VEL
LIN {X 0,Y 545.085,Z 214.087,A -85,B 0,C 180,E1 -3661.507,E2 -3661.507} C_VEL
LIN {X 0,Y 545.117,Z 214.186,A -85,B 0,C 180,E1 -3664.487,E2 -3664.487} C_VEL
LIN {X 0,Y 546.026,Z 219.885,A -85,B 0,C 180,E1 -3665.677,E2 -3665.677} C_VEL
LIN {X 0,Y 545.658,Z 235.412,A -85,B 0,C 180,E1 -3668.663,E2 -3668.663} C_VEL
LIN {X 0,Y 545.453,Z 249,A -85,B 0,C 180,E1 -3671.209,E2 -3671.209} C_VEL
LIN {X 0,Y 545.286,Z 263.623,A -85,B 0,C 180,E1 -3673.913,E2 -3673.913} C_VEL
LIN {X 0,Y 545.156,Z 272.133,A -85,B 0,C 180,E1 -3675.433,E2 -3675.433} C_VEL
LIN {X 0,Y 546.524,Z 281.026,A -85,B 0,C 180,E1 -3675.613,E2 -3675.613} C_VEL
LIN {X 0,Y 546.243,Z 376.907,A -85,B 0,C 180,E1 -3676.893,E2 -3676.893} C_VEL
LIN {X 0,Y 546.114,Z 386.805,A -85,B 0,C 180,E1 -3677.103,E2 -3677.103} C_VEL
LIN {X 0,Y 546.013,Z 396.785,A -85,B 0,C 180,E1 -3677.408,E2 -3677.408} C_VEL
LIN {X 0,Y 545.856,Z 406.144,A -85,B 0,C 180,E1 -3677.782,E2 -3677.782} C_VEL
LIN {X 0,Y 545.667,Z 416.454,A -85,B 0,C 180,E1 -3678.306,E2 -3678.306} C_VEL
LIN {X 0,Y 545.529,Z 425.291,A -85,B 0,C 180,E1 -3678.858,E2 -3678.858} C_VEL
LIN {X 0,Y 545.385,Z 434.023,A -85,B 0,C 180,E1 -3679.513,E2 -3679.513} C_VEL
LIN {X 0,Y 545.224,Z 441.421,A -85,B 0,C 180,E1 -3680.166,E2 -3680.166} C_VEL
LIN {X 0,Y 545.076,Z 448.642,A -85,B 0,C 180,E1 -3680.912,E2 -3680.912} C_VEL
LIN {X 0,Y 544.956,Z 454.844,A -85,B 0,C 180,E1 -3681.658,E2 -3681.658} C_VEL
LIN {X 0,Y 544.836,Z 461.381,A -85,B 0,C 180,E1 -3682.589,E2 -3682.589} C_VEL
LIN {X 0,Y 544.76,Z 466.255,A -85,B 0,C 180,E1 -3683.408,E2 -3683.408} C_VEL
LIN {X 0,Y 544.739,Z 471.328,A -85,B 0,C 180,E1 -3684.447,E2 -3684.447} C_VEL
LIN {X 0,Y 544.664,Z 475.624,A -85,B 0,C 180,E1 -3685.56,E2 -3685.56} C_VEL
LIN {X 0,Y 544.669,Z 477.972,A -85,B 0,C 180,E1 -3686.301,E2 -3686.301} C_VEL
LIN {X 0,Y 544.65,Z 479.758,A -85,B 0,C 180,E1 -3687.041,E2 -3687.041} C_VEL
LIN {X 0,Y 544.546,Z 482.183,A -85,B 0,C 180,E1 -3688.521,E2 -3688.521} C_VEL
LIN {X 0,Y 544.542,Z 482.766,A -85,B 0,C 180,E1 -3689.261,E2 -3689.261} C_VEL
LIN {X 0,Y 544.542,Z 482.766,A -85,B 0,C 180,E1 -3690.739,E2 -3690.739} C_VEL
LIN {X 0,Y 544.546,Z 482.183,A -85,B 0,C 180,E1 -3691.479,E2 -3691.479} C_VEL
LIN {X 0,Y 544.65,Z 479.758,A -85,B 0,C 180,E1 -3692.959,E2 -3692.959} C_VEL
LIN {X 0,Y 544.684,Z 476.832,A -85,B 0,C 180,E1 -3694.069,E2 -3694.069} C_VEL
LIN {X 0,Y 544.653,Z 472.872,A -85,B 0,C 180,E1 -3695.182,E2 -3695.182} C_VEL
LIN {X 0,Y 544.759,Z 468.63,A -85,B 0,C 180,E1 -3696.128,E2 -3696.128} C_VEL
LIN {X 0,Y 544.79,Z 463.688,A -85,B 0,C 180,E1 -3697.039,E2 -3697.039} C_VEL
LIN {X 0,Y 544.916,Z 457.596,A -85,B 0,C 180,E1 -3697.97,E2 -3697.97} C_VEL
LIN {X 0,Y 545,Z 451.896,A -85,B 0,C 180,E1 -3698.715,E2 -3698.715} C_VEL
LIN {X 0,Y 545.174,Z 443.34,A -85,B 0,C 180,E1 -3699.647,E2 -3699.647} C_VEL
LIN {X 0,Y 545.35,Z 435.158,A -85,B 0,C 180,E1 -3700.394,E2 -3700.394} C_VEL
LIN {X 0,Y 545.504,Z 426.643,A -85,B 0,C 180,E1 -3701.049,E2 -3701.049} C_VEL
LIN {X 0,Y 545.677,Z 418.185,A -85,B 0,C 180,E1 -3701.594,E2 -3701.594} C_VEL
LIN {X 0,Y 545.825,Z 409.167,A -85,B 0,C 180,E1 -3702.077,E2 -3702.077} C_VEL
LIN {X 0,Y 545.97,Z 399.361,A -85,B 0,C 180,E1 -3702.499,E2 -3702.499} C_VEL
LIN {X 0,Y 546.107,Z 389.429,A -85,B 0,C 180,E1 -3702.826,E2 -3702.826} C_VEL
LIN {X 0,Y 546.197,Z 379.57,A -85,B 0,C 180,E1 -3703.06,E2 -3703.06} C_VEL
LIN {X 0,Y 546.349,Z 354.96,A -85,B 0,C 180,E1 -3703.412,E2 -3703.412} C_VEL
LIN {X 0,Y 546.381,Z 279.325,A -85,B 0,C 180,E1 -3704.413,E2 -3704.413} C_VEL
LIN {X 0,Y 545.156,Z 272.129,A -85,B 0,C 180,E1 -3704.567,E2 -3704.567} C_VEL
LIN {X 0,Y 545.321,Z 258.403,A -85,B 0,C 180,E1 -3707.049,E2 -3707.049} C_VEL
LIN {X 0,Y 545.597,Z 243.09,A -85,B 0,C 180,E1 -3709.891,E2 -3709.891} C_VEL
LIN {X 0,Y 545.818,Z 227.171,A -85,B 0,C 180,E1 -3712.923,E2 -3712.923} C_VEL
LIN {X 0,Y 545.914,Z 218.869,A -85,B 0,C 180,E1 -3714.531,E2 -3714.531} C_VEL
LIN {X 0,Y 545.106,Z 214.11,A -85,B 0,C 180,E1 -3715.538,E2 -3715.538} C_VEL
LIN {X 0,Y 545.076,Z 214.086,A -85,B 0,C 180,E1 -3718.745,E2 -3718.745} C_VEL
LIN {X 0,Y 545.06,Z 214.092,A -85,B 0,C 180,E1 -3721.678,E2 -3721.678} C_VEL
LIN {X 0,Y 545.064,Z 214.085,A -85,B 0,C 180,E1 -3724.564,E2 -3724.564} C_VEL
LIN {X 0,Y 545.038,Z 214.089,A -85,B 0,C 180,E1 -3727.304,E2 -3727.304} C_VEL
LIN {X 0,Y 545.07,Z 214.083,A -85,B 0,C 180,E1 -3730.142,E2 -3730.142} C_VEL
LIN {X 0,Y 545.08,Z 214.084,A -85,B 0,C 180,E1 -3733.106,E2 -3733.106} C_VEL
LIN {X 0,Y 545.068,Z 214.086,A -85,B 0,C 180,E1 -3736.224,E2 -3736.224} C_VEL
LIN {X 0,Y 545.082,Z 214.082,A -85,B 0,C 180,E1 -3738.885,E2 -3738.885} C_VEL
LIN {X 0,Y 545.053,Z 214.092,A -85,B 0,C 180,E1 -3741.762,E2 -3741.762} C_VEL
LIN {X 0,Y 545.036,Z 214.086,A -85,B 0,C 180,E1 -3744.531,E2 -3744.531} C_VEL
LIN {X 0,Y 545.066,Z 214.086,A -85,B 0,C 180,E1 -3747.211,E2 -3747.211} C_VEL
LIN {X 0,Y 545.061,Z 214.088,A -85,B 0,C 180,E1 -3749.81,E2 -3749.81} C_VEL
LIN {X 0,Y 545.081,Z 214.078,A -85,B 0,C 180,E1 -3752.343,E2 -3752.343} C_VEL
LIN {X 0,Y 545.117,Z 214.077,A -85,B 0,C 180,E1 -3754.82,E2 -3754.82} C_VEL
LIN {X 0,Y 545.038,Z 214.096,A -85,B 0,C 180,E1 -3757.242,E2 -3757.242} C_VEL
LIN {X 0,Y 545.116,Z 214.074,A -85,B 0,C 180,E1 -3760.414,E2 -3760.414} C_VEL
LIN {X 0,Y 545.065,Z 214.086,A -85,B 0,C 180,E1 -3763.521,E2 -3763.521} C_VEL
LIN {X 0,Y 545.094,Z 214.081,A -85,B 0,C 180,E1 -3765.82,E2 -3765.82} C_VEL
LIN {X 0,Y 545.118,Z 214.082,A -85,B 0,C 180,E1 -3768.849,E2 -3768.849} C_VEL
LIN {X 0,Y 545.098,Z 214.076,A -85,B 0,C 180,E1 -3771.846,E2 -3771.846} C_VEL
LIN {X 0,Y 545.203,Z 214.075,A -85,B 0,C 180,E1 -3774.823,E2 -3774.823} C_VEL
LIN {X 0,Y 545.196,Z 214.066,A -85,B 0,C 180,E1 -3777.783,E2 -3777.783} C_VEL
LIN {X 0,Y 545.214,Z 214.066,A -85,B 0,C 180,E1 -3780.738,E2 -3780.738} C_VEL
LIN {X 0,Y 545.17,Z 214.077,A -85,B 0,C 180,E1 -3782.955,E2 -3782.955} C_VEL
LIN {X 0,Y 545.171,Z 214.071,A -85,B 0,C 180,E1 -3785.919,E2 -3785.919} C_VEL
LIN {X 0,Y 545.12,Z 214.075,A -85,B 0,C 180,E1 -3788.9,E2 -3788.9} C_VEL
LIN {X 0,Y 545.133,Z 214.073,A -85,B 0,C 180,E1 -3791.904,E2 -3791.904} C_VEL
LIN {X 0,Y 545.084,Z 214.085,A -85,B 0,C 180,E1 -3794.943,E2 -3794.943} C_VEL
LIN {X 0,Y 545.077,Z 214.083,A -85,B 0,C 180,E1 -3798.025,E2 -3798.025} C_VEL
LIN {X 0,Y 545.093,Z 214.084,A -85,B 0,C 180,E1 -3800.372,E2 -3800.372} C_VEL
LIN {X 0,Y 545.077,Z 214.083,A -85,B 0,C 180,E1 -3803.559,E2 -3803.559} C_VEL
LIN {X 0,Y 545.077,Z 214.086,A -85,B 0,C 180,E1 -3806,E2 -3806} C_VEL
LIN {X 0,Y 545.086,Z 214.082,A -85,B 0,C 180,E1 -3808.748,E2 -3808.748} C_VEL
LIN {X 0,Y 545.056,Z 214.088,A -85,B 0,C 180,E1 -3811.679,E2 -3811.679} C_VEL
LIN {X 0,Y 545.073,Z 214.083,A -85,B 0,C 180,E1 -3814.563,E2 -3814.563} C_VEL
LIN {X 0,Y 545.061,Z 214.085,A -85,B 0,C 180,E1 -3817.008,E2 -3817.008} C_VEL
LIN {X 0,Y 544.354,Z 214.178,A -85,B 0,C 180,E1 -3817.625,E2 -3817.625} C_VEL
LIN {X 0,Y 541.492,Z 214.533,A -85,B 0,C 180,E1 -3818.626,E2 -3818.626} C_VEL
LIN {X 0,Y 539.106,Z 214.83,A -85,B 0,C 180,E1 -3819.431,E2 -3819.431} C_VEL
LIN {X 0,Y 538.095,Z 214.957,A -85,B 0,C 180,E1 -3820.053,E2 -3820.053} C_VEL
LIN {X 0,Y 538.019,Z 214.961,A -85,B 0,C 180,E1 -3820.264,E2 -3820.264} C_VEL
LIN {X 0,Y 538.03,Z 214.961,A -85,B 0,C 180,E1 -3822.988,E2 -3822.988} C_VEL
LIN {X 0,Y 538.027,Z 214.962,A -85,B 0,C 180,E1 -3825.925,E2 -3825.925} C_VEL
LIN {X 0,Y 538.075,Z 214.949,A -85,B 0,C 180,E1 -3829.249,E2 -3829.249} C_VEL
LIN {X 0,Y 537.992,Z 214.97,A -85,B 0,C 180,E1 -3832.122,E2 -3832.122} C_VEL
LIN {X 0,Y 538.008,Z 214.959,A -85,B 0,C 180,E1 -3834.917,E2 -3834.917} C_VEL
LIN {X 0,Y 538.029,Z 214.968,A -85,B 0,C 180,E1 -3837.618,E2 -3837.618} C_VEL
LIN {X 0,Y 538.015,Z 214.959,A -85,B 0,C 180,E1 -3840.239,E2 -3840.239} C_VEL
LIN {X 0,Y 538.063,Z 214.958,A -85,B 0,C 180,E1 -3842.796,E2 -3842.796} C_VEL
LIN {X 0,Y 538.045,Z 214.966,A -85,B 0,C 180,E1 -3845.293,E2 -3845.293} C_VEL
LIN {X 0,Y 538.019,Z 214.963,A -85,B 0,C 180,E1 -3848.546,E2 -3848.546} C_VEL
LIN {X 0,Y 538.035,Z 214.964,A -85,B 0,C 180,E1 -3850.94,E2 -3850.94} C_VEL
LIN {X 0,Y 538.022,Z 214.971,A -85,B 0,C 180,E1 -3853.299,E2 -3853.299} C_VEL
LIN {X 0,Y 538.061,Z 214.963,A -85,B 0,C 180,E1 -3855.631,E2 -3855.631} C_VEL
LIN {X 0,Y 538.075,Z 214.959,A -85,B 0,C 180,E1 -3858.702,E2 -3858.702} C_VEL
LIN {X 0,Y 538.084,Z 214.958,A -85,B 0,C 180,E1 -3861.74,E2 -3861.74} C_VEL
LIN {X 0,Y 538.163,Z 214.95,A -85,B 0,C 180,E1 -3864.755,E2 -3864.755} C_VEL
LIN {X 0,Y 538.168,Z 214.946,A -85,B 0,C 180,E1 -3867.755,E2 -3867.755} C_VEL
LIN {X 0,Y 538.18,Z 214.949,A -85,B 0,C 180,E1 -3870.748,E2 -3870.748} C_VEL
LIN {X 0,Y 538.136,Z 214.957,A -85,B 0,C 180,E1 -3872.994,E2 -3872.994} C_VEL
LIN {X 0,Y 538.132,Z 214.95,A -85,B 0,C 180,E1 -3875.997,E2 -3875.997} C_VEL
LIN {X 0,Y 538.069,Z 214.964,A -85,B 0,C 180,E1 -3879.018,E2 -3879.018} C_VEL
LIN {X 0,Y 538.08,Z 214.957,A -85,B 0,C 180,E1 -3882.063,E2 -3882.063} C_VEL
LIN {X 0,Y 538.042,Z 214.964,A -85,B 0,C 180,E1 -3885.144,E2 -3885.144} C_VEL
LIN {X 0,Y 538.029,Z 214.966,A -85,B 0,C 180,E1 -3888.27,E2 -3888.27} C_VEL
LIN {X 0,Y 538.036,Z 214.969,A -85,B 0,C 180,E1 -3890.651,E2 -3890.651} C_VEL
LIN {X 0,Y 538.001,Z 214.967,A -85,B 0,C 180,E1 -3893.888,E2 -3893.888} C_VEL
LIN {X 0,Y 538.04,Z 214.968,A -85,B 0,C 180,E1 -3896.367,E2 -3896.367} C_VEL
LIN {X 0,Y 538.028,Z 214.957,A -85,B 0,C 180,E1 -3898.934,E2 -3898.934} C_VEL
LIN {X 0,Y 538.025,Z 214.965,A -85,B 0,C 180,E1 -3901.891,E2 -3901.891} C_VEL
LIN {X 0,Y 538.022,Z 214.961,A -85,B 0,C 180,E1 -3904.62,E2 -3904.62} C_VEL
LIN {X 0,Y 538.006,Z 214.964,A -85,B 0,C 180,E1 -3907.171,E2 -3907.171} C_VEL
LIN {X 0,Y 538.051,Z 214.961,A -85,B 0,C 180,E1 -3909.794,E2 -3909.794} C_VEL
LIN {X 0,Y 538.015,Z 214.956,A -85,B 0,C 180,E1 -3912.786,E2 -3912.786} C_VEL
LIN {X 0,Y 538.029,Z 214.959,A -85,B 0,C 180,E1 -3915.141,E2 -3915.141} C_VEL
LIN {X 0,Y 538.038,Z 214.963,A -85,B 0,C 180,E1 -3918.228,E2 -3918.228} C_VEL
LIN {X 0,Y 538.013,Z 214.963,A -85,B 0,C 180,E1 -3921.17,E2 -3921.17} C_VEL
LIN {X 0,Y 538.021,Z 214.965,A -85,B 0,C 180,E1 -3924.084,E2 -3924.084} C_VEL
LIN {X 0,Y 538.028,Z 214.959,A -85,B 0,C 180,E1 -3926.728,E2 -3926.728} C_VEL
LIN {X 0,Y 538.023,Z 214.967,A -85,B 0,C 180,E1 -3929.557,E2 -3929.557} C_VEL
LIN {X 0,Y 538.037,Z 214.96,A -85,B 0,C 180,E1 -3931.951,E2 -3931.951} C_VEL
LIN {X 0,Y 538.069,Z 214.955,A -85,B 0,C 180,E1 -3934.468,E2 -3934.468} C_VEL
LIN {X 0,Y 537.991,Z 214.972,A -85,B 0,C 180,E1 -3937.739,E2 -3937.739} C_VEL
LIN {X 0,Y 538.077,Z 214.95,A -85,B 0,C 180,E1 -3940.148,E2 -3940.148} C_VEL
LIN {X 0,Y 538.023,Z 214.964,A -85,B 0,C 180,E1 -3943.299,E2 -3943.299} C_VEL
LIN {X 0,Y 538.062,Z 214.963,A -85,B 0,C 180,E1 -3945.631,E2 -3945.631} C_VEL
LIN {X 0,Y 538.076,Z 214.952,A -85,B 0,C 180,E1 -3948.702,E2 -3948.702} C_VEL
LIN {X 0,Y 538.085,Z 214.955,A -85,B 0,C 180,E1 -3951.74,E2 -3951.74} C_VEL
LIN {X 0,Y 538.162,Z 214.946,A -85,B 0,C 180,E1 -3954.755,E2 -3954.755} C_VEL
LIN {X 0,Y 538.17,Z 214.941,A -85,B 0,C 180,E1 -3957.755,E2 -3957.755} C_VEL
LIN {X 0,Y 538.18,Z 214.937,A -85,B 0,C 180,E1 -3960.749,E2 -3960.749} C_VEL
LIN {X 0,Y 538.136,Z 214.952,A -85,B 0,C 180,E1 -3962.995,E2 -3962.995} C_VEL
LIN {X 0,Y 538.12,Z 214.949,A -85,B 0,C 180,E1 -3965.998,E2 -3965.998} C_VEL
LIN {X 0,Y 538.055,Z 214.957,A -85,B 0,C 180,E1 -3969.018,E2 -3969.018} C_VEL
LIN {X 0,Y 538.083,Z 214.951,A -85,B 0,C 180,E1 -3972.063,E2 -3972.063} C_VEL
LIN {X 0,Y 538.045,Z 214.962,A -85,B 0,C 180,E1 -3975.144,E2 -3975.144} C_VEL
LIN {X 0,Y 538.024,Z 214.957,A -85,B 0,C 180,E1 -3978.271,E2 -3978.271} C_VEL
LIN {X 0,Y 538.037,Z 214.962,A -85,B 0,C 180,E1 -3980.652,E2 -3980.652} C_VEL
LIN {X 0,Y 538.003,Z 214.964,A -85,B 0,C 180,E1 -3983.889,E2 -3983.889} C_VEL
LIN {X 0,Y 538.042,Z 214.96,A -85,B 0,C 180,E1 -3986.367,E2 -3986.367} C_VEL
LIN {X 0,Y 538.03,Z 214.965,A -85,B 0,C 180,E1 -3988.934,E2 -3988.934} C_VEL
LIN {X 0,Y 538.01,Z 214.964,A -85,B 0,C 180,E1 -3991.887,E2 -3991.887} C_VEL
LIN {X 0,Y 538.01,Z 214.968,A -85,B 0,C 180,E1 -3994.618,E2 -3994.618} C_VEL
LIN {X 0,Y 538.005,Z 214.965,A -85,B 0,C 180,E1 -3997.17,E2 -3997.17} C_VEL
LIN {X 0,Y 538.023,Z 214.961,A -85,B 0,C 180,E1 -3999.797,E2 -3999.797} C_VEL
LIN {X 0,Y 538.02,Z 214.965,A -85,B 0,C 180,E1 -4002.786,E2 -4002.786} C_VEL
LIN {X 0,Y 538.008,Z 214.963,A -85,B 0,C 180,E1 -4005.138,E2 -4005.138} C_VEL
LIN {X 0,Y 538.032,Z 214.965,A -85,B 0,C 180,E1 -4008.227,E2 -4008.227} C_VEL
LIN {X 0,Y 538.016,Z 214.962,A -85,B 0,C 180,E1 -4011.17,E2 -4011.17} C_VEL
LIN {X 0,Y 537.996,Z 214.969,A -85,B 0,C 180,E1 -4014.089,E2 -4014.089} C_VEL
LIN {X 0,Y 538.033,Z 214.961,A -85,B 0,C 180,E1 -4016.728,E2 -4016.728} C_VEL
LIN {X 0,Y 538.029,Z 214.966,A -85,B 0,C 180,E1 -4019.557,E2 -4019.557} C_VEL
LIN {X 0,Y 538.032,Z 214.966,A -85,B 0,C 180,E1 -4022.654,E2 -4022.654} C_VEL
LIN {X 0,Y 538.071,Z 215.154,A -85,B 0,C 180,E1 -4024.358,E2 -4024.358} C_VEL
LIN {X 0,Y 539.076,Z 221.41,A -85,B 0,C 180,E1 -4025.663,E2 -4025.663} C_VEL
LIN {X 0,Y 538.712,Z 238.409,A -85,B 0,C 180,E1 -4028.976,E2 -4028.976} C_VEL
LIN {X 0,Y 538.452,Z 253.049,A -85,B 0,C 180,E1 -4031.745,E2 -4031.745} C_VEL
LIN {X 0,Y 538.146,Z 269.679,A -85,B 0,C 180,E1 -4034.859,E2 -4034.859} C_VEL
LIN {X 0,Y 538.137,Z 271.942,A -85,B 0,C 180,E1 -4035.24,E2 -4035.24} C_VEL
LIN {X 0,Y 539.663,Z 281.867,A -85,B 0,C 180,E1 -4035.44,E2 -4035.44} C_VEL
LIN {X 0,Y 539.33,Z 376.714,A -85,B 0,C 180,E1 -4036.722,E2 -4036.722} C_VEL
LIN {X 0,Y 539.185,Z 387.487,A -85,B 0,C 180,E1 -4036.958,E2 -4036.958} C_VEL
LIN {X 0,Y 539.072,Z 396.592,A -85,B 0,C 180,E1 -4037.243,E2 -4037.243} C_VEL
LIN {X 0,Y 538.906,Z 405.951,A -85,B 0,C 180,E1 -4037.622,E2 -4037.622} C_VEL
LIN {X 0,Y 538.73,Z 415.592,A -85,B 0,C 180,E1 -4038.114,E2 -4038.114} C_VEL
LIN {X 0,Y 538.535,Z 425.097,A -85,B 0,C 180,E1 -4038.711,E2 -4038.711} C_VEL
LIN {X 0,Y 538.368,Z 433.83,A -85,B 0,C 180,E1 -4039.374,E2 -4039.374} C_VEL
LIN {X 0,Y 538.187,Z 441.227,A -85,B 0,C 180,E1 -4040.036,E2 -4040.036} C_VEL
LIN {X 0,Y 538.014,Z 448.448,A -85,B 0,C 180,E1 -4040.792,E2 -4040.792} C_VEL
LIN {X 0,Y 537.906,Z 454.651,A -85,B 0,C 180,E1 -4041.548,E2 -4041.548} C_VEL
LIN {X 0,Y 537.754,Z 461.187,A -85,B 0,C 180,E1 -4042.49,E2 -4042.49} C_VEL
LIN {X 0,Y 537.673,Z 466.577,A -85,B 0,C 180,E1 -4043.419,E2 -4043.419} C_VEL
LIN {X 0,Y 537.653,Z 471.176,A -85,B 0,C 180,E1 -4044.374,E2 -4044.374} C_VEL
LIN {X 0,Y 537.56,Z 475.494,A -85,B 0,C 180,E1 -4045.501,E2 -4045.501} C_VEL
LIN {X 0,Y 537.591,Z 477.858,A -85,B 0,C 180,E1 -4046.252,E2 -4046.252} C_VEL
LIN {X 0,Y 537.551,Z 479.652,A -85,B 0,C 180,E1 -4047.002,E2 -4047.002} C_VEL
LIN {X 0,Y 537.451,Z 482.089,A -85,B 0,C 180,E1 -4048.501,E2 -4048.501} C_VEL
LIN {X 0,Y 537.442,Z 482.676,A -85,B 0,C 180,E1 -4049.251,E2 -4049.251} C_VEL
LIN {X 0,Y 537.442,Z 482.676,A -85,B 0,C 180,E1 -4050.749,E2 -4050.749} C_VEL
LIN {X 0,Y 537.451,Z 482.089,A -85,B 0,C 180,E1 -4051.499,E2 -4051.499} C_VEL
LIN {X 0,Y 537.551,Z 479.652,A -85,B 0,C 180,E1 -4052.998,E2 -4052.998} C_VEL
LIN {X 0,Y 537.604,Z 476.711,A -85,B 0,C 180,E1 -4054.123,E2 -4054.123} C_VEL
LIN {X 0,Y 537.586,Z 472.727,A -85,B 0,C 180,E1 -4055.251,E2 -4055.251} C_VEL
LIN {X 0,Y 537.63,Z 467.911,A -85,B 0,C 180,E1 -4056.318,E2 -4056.318} C_VEL
LIN {X 0,Y 537.754,Z 462.343,A -85,B 0,C 180,E1 -4057.321,E2 -4057.321} C_VEL
LIN {X 0,Y 537.873,Z 456.027,A -85,B 0,C 180,E1 -4058.264,E2 -4058.264} C_VEL
LIN {X 0,Y 537.98,Z 450.075,A -85,B 0,C 180,E1 -4059.019,E2 -4059.019} C_VEL
LIN {X 0,Y 538.132,Z 443.146,A -85,B 0,C 180,E1 -4059.775,E2 -4059.775} C_VEL
LIN {X 0,Y 538.305,Z 436.1,A -85,B 0,C 180,E1 -4060.437,E2 -4060.437} C_VEL
LIN {X 0,Y 538.482,Z 427.802,A -85,B 0,C 180,E1 -4061.099,E2 -4061.099} C_VEL
LIN {X 0,Y 538.694,Z 418.055,A -85,B 0,C 180,E1 -4061.743,E2 -4061.743} C_VEL
LIN {X 0,Y 538.881,Z 407.966,A -85,B 0,C 180,E1 -4062.283,E2 -4062.283} C_VEL
LIN {X 0,Y 539.021,Z 399.168,A -85,B 0,C 180,E1 -4062.663,E2 -4062.663} C_VEL
LIN {X 0,Y 539.164,Z 389.236,A -85,B 0,C 180,E1 -4062.994,E2 -4062.994} C_VEL
LIN {X 0,Y 539.3,Z 379.378,A -85,B 0,C 180,E1 -4063.23,E2 -4063.23} C_VEL
LIN {X 0,Y 539.453,Z 354.767,A -85,B 0,C 180,E1 -4063.586,E2 -4063.586} C_VEL
LIN {X 0,Y 539.608,Z 280.704,A -85,B 0,C 180,E1 -4064.577,E2 -4064.577} C_VEL
LIN {X 0,Y 538.125,Z 271.938,A -85,B 0,C 180,E1 -4064.761,E2 -4064.761} C_VEL
LIN {X 0,Y 538.157,Z 268.69,A -85,B 0,C 180,E1 -4065.334,E2 -4065.334} C_VEL
LIN {X 0,Y 538.422,Z 252.003,A -85,B 0,C 180,E1 -4068.453,E2 -4068.453} C_VEL
LIN {X 0,Y 538.678,Z 238.409,A -85,B 0,C 180,E1 -4071.026,E2 -4071.026} C_VEL
LIN {X 0,Y 539.032,Z 222.507,A -85,B 0,C 180,E1 -4074.122,E2 -4074.122} C_VEL
LIN {X 0,Y 538.557,Z 217.715,A -85,B 0,C 180,E1 -4075.095,E2 -4075.095} C_VEL
LIN {X 0,Y 538.05,Z 214.989,A -85,B 0,C 180,E1 -4075.709,E2 -4075.709} C_VEL
LIN {X 0,Y 538.023,Z 214.968,A -85,B 0,C 180,E1 -4078.051,E2 -4078.051} C_VEL
LIN {X 0,Y 538.023,Z 214.965,A -85,B 0,C 180,E1 -4080.627,E2 -4080.627} C_VEL
LIN {X 0,Y 538.048,Z 214.96,A -85,B 0,C 180,E1 -4083.282,E2 -4083.282} C_VEL
LIN {X 0,Y 537.996,Z 214.97,A -85,B 0,C 180,E1 -4086.004,E2 -4086.004} C_VEL
LIN {X 0,Y 538.016,Z 214.962,A -85,B 0,C 180,E1 -4088.83,E2 -4088.83} C_VEL
LIN {X 0,Y 538.032,Z 214.965,A -85,B 0,C 180,E1 -4091.773,E2 -4091.773} C_VEL
LIN {X 0,Y 538.008,Z 214.963,A -85,B 0,C 180,E1 -4094.862,E2 -4094.862} C_VEL
LIN {X 0,Y 538.02,Z 214.965,A -85,B 0,C 180,E1 -4097.214,E2 -4097.214} C_VEL
LIN {X 0,Y 538.023,Z 214.961,A -85,B 0,C 180,E1 -4100.203,E2 -4100.203} C_VEL
LIN {X 0,Y 538.025,Z 214.964,A -85,B 0,C 180,E1 -4103.067,E2 -4103.067} C_VEL
LIN {X 0,Y 538.011,Z 214.963,A -85,B 0,C 180,E1 -4105.826,E2 -4105.826} C_VEL
LIN {X 0,Y 538.009,Z 214.963,A -85,B 0,C 180,E1 -4108.498,E2 -4108.498} C_VEL
LIN {X 0,Y 538.043,Z 214.964,A -85,B 0,C 180,E1 -4111.099,E2 -4111.099} C_VEL
LIN {X 0,Y 538.042,Z 214.96,A -85,B 0,C 180,E1 -4113.633,E2 -4113.633} C_VEL
LIN {X 0,Y 538.007,Z 214.963,A -85,B 0,C 180,E1 -4116.122,E2 -4116.122} C_VEL
LIN {X 0,Y 538.037,Z 214.962,A -85,B 0,C 180,E1 -4119.348,E2 -4119.348} C_VEL
LIN {X 0,Y 538.036,Z 214.955,A -85,B 0,C 180,E1 -4122.467,E2 -4122.467} C_VEL
LIN {X 0,Y 538.064,Z 214.958,A -85,B 0,C 180,E1 -4125.63,E2 -4125.63} C_VEL
LIN {X 0,Y 538.077,Z 214.956,A -85,B 0,C 180,E1 -4128.701,E2 -4128.701} C_VEL
LIN {X 0,Y 538.061,Z 214.953,A -85,B 0,C 180,E1 -4131.739,E2 -4131.739} C_VEL
LIN {X 0,Y 538.16,Z 214.951,A -85,B 0,C 180,E1 -4134.755,E2 -4134.755} C_VEL
LIN {X 0,Y 538.168,Z 214.941,A -85,B 0,C 180,E1 -4137.754,E2 -4137.754} C_VEL
LIN {X 0,Y 538.183,Z 214.941,A -85,B 0,C 180,E1 -4140.748,E2 -4140.748} C_VEL
LIN {X 0,Y 538.136,Z 214.952,A -85,B 0,C 180,E1 -4142.994,E2 -4142.994} C_VEL
LIN {X 0,Y 538.121,Z 214.95,A -85,B 0,C 180,E1 -4145.997,E2 -4145.997} C_VEL
LIN {X 0,Y 538.07,Z 214.951,A -85,B 0,C 180,E1 -4149.017,E2 -4149.017} C_VEL
LIN {X 0,Y 538.082,Z 214.953,A -85,B 0,C 180,E1 -4152.062,E2 -4152.062} C_VEL
LIN {X 0,Y 538.044,Z 214.96,A -85,B 0,C 180,E1 -4155.143,E2 -4155.143} C_VEL
LIN {X 0,Y 538.03,Z 214.964,A -85,B 0,C 180,E1 -4158.27,E2 -4158.27} C_VEL
LIN {X 0,Y 538.037,Z 214.963,A -85,B 0,C 180,E1 -4160.651,E2 -4160.651} C_VEL
LIN {X 0,Y 538,Z 214.968,A -85,B 0,C 180,E1 -4163.888,E2 -4163.888} C_VEL
LIN {X 0,Y 538.039,Z 214.961,A -85,B 0,C 180,E1 -4166.366,E2 -4166.366} C_VEL
LIN {X 0,Y 538.028,Z 214.96,A -85,B 0,C 180,E1 -4168.933,E2 -4168.933} C_VEL
LIN {X 0,Y 538.012,Z 214.968,A -85,B 0,C 180,E1 -4171.888,E2 -4171.888} C_VEL
LIN {X 0,Y 538.023,Z 214.96,A -85,B 0,C 180,E1 -4174.62,E2 -4174.62} C_VEL
LIN {X 0,Y 538.004,Z 214.964,A -85,B 0,C 180,E1 -4177.17,E2 -4177.17} C_VEL
LIN {X 0,Y 538.019,Z 214.961,A -85,B 0,C 180,E1 -4180.264,E2 -4180.264} C_VEL
LIN {X 0,Y 537.369,Z 215.041,A -85,B 0,C 180,E1 -4180.889,E2 -4180.889} C_VEL
LIN {X 0,Y 534.519,Z 215.403,A -85,B 0,C 180,E1 -4181.904,E2 -4181.904} C_VEL
LIN {X 0,Y 532.096,Z 215.707,A -85,B 0,C 180,E1 -4182.721,E2 -4182.721} C_VEL
LIN {X 0,Y 531.048,Z 215.835,A -85,B 0,C 180,E1 -4183.352,E2 -4183.352} C_VEL
LIN {X 0,Y 530.96,Z 215.844,A -85,B 0,C 180,E1 -4183.566,E2 -4183.566} C_VEL
LIN {X 0,Y 530.961,Z 215.834,A -85,B 0,C 180,E1 -4186.505,E2 -4186.505} C_VEL
LIN {X 0,Y 531.023,Z 215.831,A -85,B 0,C 180,E1 -4189.571,E2 -4189.571} C_VEL
LIN {X 0,Y 530.966,Z 215.841,A -85,B 0,C 180,E1 -4192.576,E2 -4192.576} C_VEL
LIN {X 0,Y 530.992,Z 215.836,A -85,B 0,C 180,E1 -4195.311,E2 -4195.311} C_VEL
LIN {X 0,Y 530.98,Z 215.843,A -85,B 0,C 180,E1 -4198.033,E2 -4198.033} C_VEL
LIN {X 0,Y 530.986,Z 215.833,A -85,B 0,C 180,E1 -4200.874,E2 -4200.874} C_VEL
LIN {X 0,Y 531.003,Z 215.842,A -85,B 0,C 180,E1 -4203.256,E2 -4203.256} C_VEL
LIN {X 0,Y 530.982,Z 215.843,A -85,B 0,C 180,E1 -4205.96,E2 -4205.96} C_VEL
LIN {X 0,Y 530.997,Z 215.842,A -85,B 0,C 180,E1 -4209.062,E2 -4209.062} C_VEL
LIN {X 0,Y 531.013,Z 215.837,A -85,B 0,C 180,E1 -4212.278,E2 -4212.278} C_VEL
LIN {X 0,Y 531.037,Z 215.84,A -85,B 0,C 180,E1 -4215.436,E2 -4215.436} C_VEL
LIN {X 0,Y 531.034,Z 215.835,A -85,B 0,C 180,E1 -4218.55,E2 -4218.55} C_VEL
LIN {X 0,Y 531.054,Z 215.835,A -85,B 0,C 180,E1 -4221.629,E2 -4221.629} C_VEL
LIN {X 0,Y 531.122,Z 215.826,A -85,B 0,C 180,E1 -4224.685,E2 -4224.685} C_VEL
LIN {X 0,Y 531.139,Z 215.822,A -85,B 0,C 180,E1 -4227.725,E2 -4227.725} C_VEL
LIN {X 0,Y 531.15,Z 215.825,A -85,B 0,C 180,E1 -4230.758,E2 -4230.758} C_VEL
LIN {X 0,Y 531.102,Z 215.832,A -85,B 0,C 180,E1 -4233.034,E2 -4233.034} C_VEL
LIN {X 0,Y 531.09,Z 215.828,A -85,B 0,C 180,E1 -4236.077,E2 -4236.077} C_VEL
LIN {X 0,Y 531.029,Z 215.839,A -85,B 0,C 180,E1 -4239.138,E2 -4239.138} C_VEL
LIN {X 0,Y 531.038,Z 215.836,A -85,B 0,C 180,E1 -4242.225,E2 -4242.225} C_VEL
LIN {X 0,Y 530.992,Z 215.84,A -85,B 0,C 180,E1 -4245.35,E2 -4245.35} C_VEL
LIN {X 0,Y 530.988,Z 215.846,A -85,B 0,C 180,E1 -4248.521,E2 -4248.521} C_VEL
LIN {X 0,Y 530.997,Z 215.842,A -85,B 0,C 180,E1 -4250.938,E2 -4250.938} C_VEL
LIN {X 0,Y 530.968,Z 215.846,A -85,B 0,C 180,E1 -4254.225,E2 -4254.225} C_VEL
LIN {X 0,Y 531.003,Z 215.842,A -85,B 0,C 180,E1 -4256.744,E2 -4256.744} C_VEL
LIN {X 0,Y 530.979,Z 215.833,A -85,B 0,C 180,E1 -4259.323,E2 -4259.323} C_VEL
LIN {X 0,Y 530.977,Z 215.845,A -85,B 0,C 180,E1 -4262.103,E2 -4262.103} C_VEL
LIN {X 0,Y 530.979,Z 215.835,A -85,B 0,C 180,E1 -4264.853,E2 -4264.853} C_VEL
LIN {X 0,Y 530.964,Z 215.842,A -85,B 0,C 180,E1 -4267.508,E2 -4267.508} C_VEL
LIN {X 0,Y 531.023,Z 215.831,A -85,B 0,C 180,E1 -4270.429,E2 -4270.429} C_VEL
LIN {X 0,Y 530.961,Z 215.834,A -85,B 0,C 180,E1 -4273.495,E2 -4273.495} C_VEL
LIN {X 0,Y 530.963,Z 215.844,A -85,B 0,C 180,E1 -4276.506,E2 -4276.506} C_VEL
LIN {X 0,Y 530.989,Z 215.837,A -85,B 0,C 180,E1 -4279.568,E2 -4279.568} C_VEL
LIN {X 0,Y 530.966,Z 215.842,A -85,B 0,C 180,E1 -4282.577,E2 -4282.577} C_VEL
LIN {X 0,Y 530.993,Z 215.835,A -85,B 0,C 180,E1 -4285.311,E2 -4285.311} C_VEL
LIN {X 0,Y 530.969,Z 215.847,A -85,B 0,C 180,E1 -4288.033,E2 -4288.033} C_VEL
LIN {X 0,Y 530.986,Z 215.837,A -85,B 0,C 180,E1 -4290.874,E2 -4290.874} C_VEL
LIN {X 0,Y 530.999,Z 215.832,A -85,B 0,C 180,E1 -4293.257,E2 -4293.257} C_VEL
LIN {X 0,Y 530.982,Z 215.844,A -85,B 0,C 180,E1 -4295.961,E2 -4295.961} C_VEL
LIN {X 0,Y 530.998,Z 215.837,A -85,B 0,C 180,E1 -4299.063,E2 -4299.063} C_VEL
LIN {X 0,Y 531.015,Z 215.832,A -85,B 0,C 180,E1 -4302.278,E2 -4302.278} C_VEL
LIN {X 0,Y 531.039,Z 215.84,A -85,B 0,C 180,E1 -4305.437,E2 -4305.437} C_VEL
LIN {X 0,Y 531.036,Z 215.828,A -85,B 0,C 180,E1 -4308.55,E2 -4308.55} C_VEL
LIN {X 0,Y 531.055,Z 215.832,A -85,B 0,C 180,E1 -4311.63,E2 -4311.63} C_VEL
LIN {X 0,Y 531.121,Z 215.823,A -85,B 0,C 180,E1 -4314.686,E2 -4314.686} C_VEL
LIN {X 0,Y 531.141,Z 215.816,A -85,B 0,C 180,E1 -4317.725,E2 -4317.725} C_VEL
LIN {X 0,Y 531.15,Z 215.812,A -85,B 0,C 180,E1 -4320.759,E2 -4320.759} C_VEL
LIN {X 0,Y 531.103,Z 215.829,A -85,B 0,C 180,E1 -4323.035,E2 -4323.035} C_VEL
LIN {X 0,Y 531.074,Z 215.826,A -85,B 0,C 180,E1 -4326.078,E2 -4326.078} C_VEL
LIN {X 0,Y 531.017,Z 215.832,A -85,B 0,C 180,E1 -4329.139,E2 -4329.139} C_VEL
LIN {X 0,Y 531.04,Z 215.829,A -85,B 0,C 180,E1 -4332.225,E2 -4332.225} C_VEL
LIN {X 0,Y 530.995,Z 215.838,A -85,B 0,C 180,E1 -4335.35,E2 -4335.35} C_VEL
LIN {X 0,Y 530.984,Z 215.836,A -85,B 0,C 180,E1 -4338.522,E2 -4338.522} C_VEL
LIN {X 0,Y 530.999,Z 215.842,A -85,B 0,C 180,E1 -4340.938,E2 -4340.938} C_VEL
LIN {X 0,Y 530.972,Z 215.842,A -85,B 0,C 180,E1 -4344.225,E2 -4344.225} C_VEL
LIN {X 0,Y 531.002,Z 215.837,A -85,B 0,C 180,E1 -4346.744,E2 -4346.744} C_VEL
LIN {X 0,Y 530.981,Z 215.839,A -85,B 0,C 180,E1 -4349.323,E2 -4349.323} C_VEL
LIN {X 0,Y 530.965,Z 215.843,A -85,B 0,C 180,E1 -4352.1,E2 -4352.1} C_VEL
LIN {X 0,Y 530.969,Z 215.843,A -85,B 0,C 180,E1 -4354.851,E2 -4354.851} C_VEL
LIN {X 0,Y 530.966,Z 215.841,A -85,B 0,C 180,E1 -4357.508,E2 -4357.508} C_VEL
LIN {X 0,Y 530.982,Z 215.844,A -85,B 0,C 180,E1 -4360.433,E2 -4360.433} C_VEL
LIN {X 0,Y 530.966,Z 215.841,A -85,B 0,C 180,E1 -4363.495,E2 -4363.495} C_VEL
LIN {X 0,Y 530.966,Z 215.846,A -85,B 0,C 180,E1 -4366.506,E2 -4366.506} C_VEL
LIN {X 0,Y 530.983,Z 215.834,A -85,B 0,C 180,E1 -4369.567,E2 -4369.567} C_VEL
LIN {X 0,Y 530.969,Z 215.843,A -85,B 0,C 180,E1 -4372.577,E2 -4372.577} C_VEL
LIN {X 0,Y 530.984,Z 215.838,A -85,B 0,C 180,E1 -4375.31,E2 -4375.31} C_VEL
LIN {X 0,Y 530.969,Z 215.846,A -85,B 0,C 180,E1 -4378.032,E2 -4378.032} C_VEL
LIN {X 0,Y 530.99,Z 215.841,A -85,B 0,C 180,E1 -4380.875,E2 -4380.875} C_VEL
LIN {X 0,Y 531.019,Z 215.93,A -85,B 0,C 180,E1 -4384.155,E2 -4384.155} C_VEL
LIN {X 0,Y 532.008,Z 221.656,A -85,B 0,C 180,E1 -4385.395,E2 -4385.395} C_VEL
LIN {X 0,Y 531.81,Z 233.149,A -85,B 0,C 180,E1 -4387.679,E2 -4387.679} C_VEL
LIN {X 0,Y 531.568,Z 246.645,A -85,B 0,C 180,E1 -4390.297,E2 -4390.297} C_VEL
LIN {X 0,Y 531.272,Z 260.228,A -85,B 0,C 180,E1 -4392.882,E2 -4392.882} C_VEL
LIN {X 0,Y 531.101,Z 271.484,A -85,B 0,C 180,E1 -4395.018,E2 -4395.018} C_VEL
LIN {X 0,Y 531.459,Z 274.198,A -85,B 0,C 180,E1 -4395.108,E2 -4395.108} C_VEL
LIN {X 0,Y 532.799,Z 283.186,A -85,B 0,C 180,E1 -4395.269,E2 -4395.269} C_VEL
LIN {X 0,Y 532.427,Z 376.522,A -85,B 0,C 180,E1 -4396.547,E2 -4396.547} C_VEL
LIN {X 0,Y 532.27,Z 387.294,A -85,B 0,C 180,E1 -4396.786,E2 -4396.786} C_VEL
LIN {X 0,Y 532.126,Z 396.398,A -85,B 0,C 180,E1 -4397.074,E2 -4397.074} C_VEL
LIN {X 0,Y 531.943,Z 406.765,A -85,B 0,C 180,E1 -4397.506,E2 -4397.506} C_VEL
LIN {X 0,Y 531.73,Z 415.839,A -85,B 0,C 180,E1 -4397.981,E2 -4397.981} C_VEL
LIN {X 0,Y 531.536,Z 424.903,A -85,B 0,C 180,E1 -4398.561,E2 -4398.561} C_VEL
LIN {X 0,Y 531.339,Z 433.635,A -85,B 0,C 180,E1 -4399.232,E2 -4399.232} C_VEL
LIN {X 0,Y 531.144,Z 441.033,A -85,B 0,C 180,E1 -4399.903,E2 -4399.903} C_VEL
LIN {X 0,Y 530.983,Z 448.254,A -85,B 0,C 180,E1 -4400.669,E2 -4400.669} C_VEL
LIN {X 0,Y 530.862,Z 454.457,A -85,B 0,C 180,E1 -4401.435,E2 -4401.435} C_VEL
LIN {X 0,Y 530.688,Z 460.993,A -85,B 0,C 180,E1 -4402.39,E2 -4402.39} C_VEL
LIN {X 0,Y 530.569,Z 466.965,A -85,B 0,C 180,E1 -4403.447,E2 -4403.447} C_VEL
LIN {X 0,Y 530.572,Z 470.983,A -85,B 0,C 180,E1 -4404.299,E2 -4404.299} C_VEL
LIN {X 0,Y 530.458,Z 475.301,A -85,B 0,C 180,E1 -4405.441,E2 -4405.441} C_VEL
LIN {X 0,Y 530.516,Z 477.666,A -85,B 0,C 180,E1 -4406.202,E2 -4406.202} C_VEL
LIN {X 0,Y 530.457,Z 479.46,A -85,B 0,C 180,E1 -4406.962,E2 -4406.962} C_VEL
LIN {X 0,Y 530.361,Z 481.896,A -85,B 0,C 180,E1 -4408.481,E2 -4408.481} C_VEL
LIN {X 0,Y 530.345,Z 482.483,A -85,B 0,C 180,E1 -4409.241,E2 -4409.241} C_VEL
LIN {X 0,Y 530.345,Z 482.483,A -85,B 0,C 180,E1 -4410.759,E2 -4410.759} C_VEL
LIN {X 0,Y 530.361,Z 481.896,A -85,B 0,C 180,E1 -4411.519,E2 -4411.519} C_VEL
LIN {X 0,Y 530.457,Z 479.46,A -85,B 0,C 180,E1 -4413.038,E2 -4413.038} C_VEL
LIN {X 0,Y 530.524,Z 476.518,A -85,B 0,C 180,E1 -4414.178,E2 -4414.178} C_VEL
LIN {X 0,Y 530.52,Z 472.534,A -85,B 0,C 180,E1 -4415.321,E2 -4415.321} C_VEL
LIN {X 0,Y 530.537,Z 468.243,A -85,B 0,C 180,E1 -4416.299,E2 -4416.299} C_VEL
LIN {X 0,Y 530.666,Z 463.305,A -85,B 0,C 180,E1 -4417.228,E2 -4417.228} C_VEL
LIN {X 0,Y 530.781,Z 457.209,A -85,B 0,C 180,E1 -4418.183,E2 -4418.183} C_VEL
LIN {X 0,Y 530.903,Z 451.508,A -85,B 0,C 180,E1 -4418.948,E2 -4418.948} C_VEL
LIN {X 0,Y 531.093,Z 442.952,A -85,B 0,C 180,E1 -4419.906,E2 -4419.906} C_VEL
LIN {X 0,Y 531.334,Z 434.771,A -85,B 0,C 180,E1 -4420.672,E2 -4420.672} C_VEL
LIN {X 0,Y 531.53,Z 426.256,A -85,B 0,C 180,E1 -4421.343,E2 -4421.343} C_VEL
LIN {X 0,Y 531.698,Z 417.861,A -85,B 0,C 180,E1 -4421.9,E2 -4421.9} C_VEL
LIN {X 0,Y 531.91,Z 407.772,A -85,B 0,C 180,E1 -4422.447,E2 -4422.447} C_VEL
LIN {X 0,Y 532.121,Z 397.687,A -85,B 0,C 180,E1 -4422.878,E2 -4422.878} C_VEL
LIN {X 0,Y 532.27,Z 388.169,A -85,B 0,C 180,E1 -4423.19,E2 -4423.19} C_VEL
LIN {X 0,Y 532.407,Z 377.853,A -85,B 0,C 180,E1 -4423.429,E2 -4423.429} C_VEL
LIN {X 0,Y 532.663,Z 302.662,A -85,B 0,C 180,E1 -4424.469,E2 -4424.469} C_VEL
LIN {X 0,Y 532.713,Z 281.417,A -85,B 0,C 180,E1 -4424.758,E2 -4424.758} C_VEL
LIN {X 0,Y 531.148,Z 272.026,A -85,B 0,C 180,E1 -4424.943,E2 -4424.943} C_VEL
LIN {X 0,Y 531.09,Z 270.631,A -85,B 0,C 180,E1 -4425.127,E2 -4425.127} C_VEL
LIN {X 0,Y 531.398,Z 255.215,A -85,B 0,C 180,E1 -4428.067,E2 -4428.067} C_VEL
LIN {X 0,Y 531.694,Z 240.368,A -85,B 0,C 180,E1 -4430.909,E2 -4430.909} C_VEL
LIN {X 0,Y 532.063,Z 223.8,A -85,B 0,C 180,E1 -4434.172,E2 -4434.172} C_VEL
LIN {X 0,Y 531.697,Z 219.658,A -85,B 0,C 180,E1 -4435.023,E2 -4435.023} C_VEL
LIN {X 0,Y 531.012,Z 215.87,A -85,B 0,C 180,E1 -4435.869,E2 -4435.869} C_VEL
LIN {X 0,Y 530.99,Z 215.841,A -85,B 0,C 180,E1 -4439.125,E2 -4439.125} C_VEL
LIN {X 0,Y 530.967,Z 215.846,A -85,B 0,C 180,E1 -4442.1,E2 -4442.1} C_VEL
LIN {X 0,Y 530.972,Z 215.84,A -85,B 0,C 180,E1 -4444.851,E2 -4444.851} C_VEL
LIN {X 0,Y 530.967,Z 215.845,A -85,B 0,C 180,E1 -4447.507,E2 -4447.507} C_VEL
LIN {X 0,Y 530.983,Z 215.834,A -85,B 0,C 180,E1 -4450.433,E2 -4450.433} C_VEL
LIN {X 0,Y 530.966,Z 215.846,A -85,B 0,C 180,E1 -4453.494,E2 -4453.494} C_VEL
LIN {X 0,Y 530.966,Z 215.841,A -85,B 0,C 180,E1 -4456.505,E2 -4456.505} C_VEL
LIN {X 0,Y 530.982,Z 215.844,A -85,B 0,C 180,E1 -4459.567,E2 -4459.567} C_VEL
LIN {X 0,Y 530.968,Z 215.841,A -85,B 0,C 180,E1 -4462.577,E2 -4462.577} C_VEL
LIN {X 0,Y 530.981,Z 215.843,A -85,B 0,C 180,E1 -4465.309,E2 -4465.309} C_VEL
LIN {X 0,Y 530.967,Z 215.842,A -85,B 0,C 180,E1 -4468.031,E2 -4468.031} C_VEL
LIN {X 0,Y 530.988,Z 215.84,A -85,B 0,C 180,E1 -4470.874,E2 -4470.874} C_VEL
LIN {X 0,Y 531.002,Z 215.837,A -85,B 0,C 180,E1 -4473.256,E2 -4473.256} C_VEL
LIN {X 0,Y 530.985,Z 215.839,A -85,B 0,C 180,E1 -4475.96,E2 -4475.96} C_VEL
LIN {X 0,Y 530.999,Z 215.842,A -85,B 0,C 180,E1 -4479.062,E2 -4479.062} C_VEL
LIN {X 0,Y 530.985,Z 215.836,A -85,B 0,C 180,E1 -4481.478,E2 -4481.478} C_VEL
LIN {X 0,Y 530.995,Z 215.838,A -85,B 0,C 180,E1 -4484.65,E2 -4484.65} C_VEL
LIN {X 0,Y 531.04,Z 215.829,A -85,B 0,C 180,E1 -4487.775,E2 -4487.775} C_VEL
LIN {X 0,Y 531.017,Z 215.832,A -85,B 0,C 180,E1 -4490.861,E2 -4490.861} C_VEL
LIN {X 0,Y 531.074,Z 215.826,A -85,B 0,C 180,E1 -4493.922,E2 -4493.922} C_VEL
LIN {X 0,Y 531.103,Z 215.829,A -85,B 0,C 180,E1 -4496.965,E2 -4496.965} C_VEL
LIN {X 0,Y 531.143,Z 215.81,A -85,B 0,C 180,E1 -4500,E2 -4500} C_VEL
LIN {X 0,Y 531.103,Z 215.828,A -85,B 0,C 180,E1 -4503.034,E2 -4503.034} C_VEL
LIN {X 0,Y 531.075,Z 215.828,A -85,B 0,C 180,E1 -4506.077,E2 -4506.077} C_VEL
LIN {X 0,Y 531.055,Z 215.832,A -85,B 0,C 180,E1 -4508.37,E2 -4508.37} C_VEL
LIN {X 0,Y 531.05,Z 215.826,A -85,B 0,C 180,E1 -4511.672,E2 -4511.672} C_VEL
LIN {X 0,Y 531.029,Z 215.835,A -85,B 0,C 180,E1 -4514.955,E2 -4514.955} C_VEL
LIN {X 0,Y 531.015,Z 215.832,A -85,B 0,C 180,E1 -4517.722,E2 -4517.722} C_VEL
LIN {X 0,Y 530.998,Z 215.837,A -85,B 0,C 180,E1 -4520.937,E2 -4520.937} C_VEL
LIN {X 0,Y 530.963,Z 215.849,A -85,B 0,C 180,E1 -4524.225,E2 -4524.225} C_VEL
LIN {X 0,Y 530.999,Z 215.832,A -85,B 0,C 180,E1 -4526.743,E2 -4526.743} C_VEL
LIN {X 0,Y 530.979,Z 215.837,A -85,B 0,C 180,E1 -4529.322,E2 -4529.322} C_VEL
LIN {X 0,Y 530.968,Z 215.849,A -85,B 0,C 180,E1 -4532.101,E2 -4532.101} C_VEL
LIN {X 0,Y 530.98,Z 215.836,A -85,B 0,C 180,E1 -4534.853,E2 -4534.853} C_VEL
LIN {X 0,Y 530.964,Z 215.843,A -85,B 0,C 180,E1 -4537.507,E2 -4537.507} C_VEL
LIN {X 0,Y 530.982,Z 215.838,A -85,B 0,C 180,E1 -4540.432,E2 -4540.432} C_VEL
LIN {X 0,Y 530.967,Z 215.842,A -85,B 0,C 180,E1 -4543.282,E2 -4543.282} C_VEL
LIN {X 0,Y 530.96,Z 215.844,A -85,B 0,C 180,E1 -4543.566,E2 -4543.566} C_VEL
LIN {X 0,Y 530.286,Z 215.929,A -85,B 0,C 180,E1 -4544.2,E2 -4544.2} C_VEL
LIN {X 0,Y 527.438,Z 216.28,A -85,B 0,C 180,E1 -4545.228,E2 -4545.228} C_VEL
LIN {X 0,Y 525.034,Z 216.577,A -85,B 0,C 180,E1 -4546.057,E2 -4546.057} C_VEL
LIN {X 0,Y 524.001,Z 216.7,A -85,B 0,C 180,E1 -4546.696,E2 -4546.696} C_VEL
LIN {X 0,Y 523.916,Z 216.71,A -85,B 0,C 180,E1 -4546.913,E2 -4546.913} C_VEL
LIN {X 0,Y 523.975,Z 216.714,A -85,B 0,C 180,E1 -4549.923,E2 -4549.923} C_VEL
LIN {X 0,Y 523.909,Z 216.72,A -85,B 0,C 180,E1 -4552.868,E2 -4552.868} C_VEL
LIN {X 0,Y 523.937,Z 216.715,A -85,B 0,C 180,E1 -4555.71,E2 -4555.71} C_VEL
LIN {X 0,Y 523.928,Z 216.718,A -85,B 0,C 180,E1 -4558.457,E2 -4558.457} C_VEL
LIN {X 0,Y 523.937,Z 216.713,A -85,B 0,C 180,E1 -4561.125,E2 -4561.125} C_VEL
LIN {X 0,Y 523.981,Z 216.715,A -85,B 0,C 180,E1 -4563.98,E2 -4563.98} C_VEL
LIN {X 0,Y 523.922,Z 216.72,A -85,B 0,C 180,E1 -4566.27,E2 -4566.27} C_VEL
LIN {X 0,Y 523.943,Z 216.718,A -85,B 0,C 180,E1 -4568.767,E2 -4568.767} C_VEL
LIN {X 0,Y 523.949,Z 216.723,A -85,B 0,C 180,E1 -4571.221,E2 -4571.221} C_VEL
LIN {X 0,Y 523.934,Z 216.723,A -85,B 0,C 180,E1 -4573.639,E2 -4573.639} C_VEL
LIN {X 0,Y 523.942,Z 216.718,A -85,B 0,C 180,E1 -4576.028,E2 -4576.028} C_VEL
LIN {X 0,Y 524.009,Z 216.71,A -85,B 0,C 180,E1 -4578.394,E2 -4578.394} C_VEL
LIN {X 0,Y 524.002,Z 216.715,A -85,B 0,C 180,E1 -4581.516,E2 -4581.516} C_VEL
LIN {X 0,Y 524.084,Z 216.703,A -85,B 0,C 180,E1 -4584.614,E2 -4584.614} C_VEL
LIN {X 0,Y 524.111,Z 216.698,A -85,B 0,C 180,E1 -4587.694,E2 -4587.694} C_VEL
LIN {X 0,Y 524.12,Z 216.701,A -85,B 0,C 180,E1 -4590.768,E2 -4590.768} C_VEL
LIN {X 0,Y 524.069,Z 216.708,A -85,B 0,C 180,E1 -4593.075,E2 -4593.075} C_VEL
LIN {X 0,Y 524.051,Z 216.705,A -85,B 0,C 180,E1 -4596.159,E2 -4596.159} C_VEL
LIN {X 0,Y 523.997,Z 216.714,A -85,B 0,C 180,E1 -4599.262,E2 -4599.262} C_VEL
LIN {X 0,Y 524,Z 216.711,A -85,B 0,C 180,E1 -4601.74,E2 -4601.74} C_VEL
LIN {X 0,Y 523.991,Z 216.716,A -85,B 0,C 180,E1 -4605.053,E2 -4605.053} C_VEL
LIN {X 0,Y 523.961,Z 216.716,A -85,B 0,C 180,E1 -4607.969,E2 -4607.969} C_VEL
LIN {X 0,Y 523.969,Z 216.72,A -85,B 0,C 180,E1 -4610.41,E2 -4610.41} C_VEL
LIN {X 0,Y 523.908,Z 216.725,A -85,B 0,C 180,E1 -4612.894,E2 -4612.894} C_VEL
LIN {X 0,Y 523.949,Z 216.716,A -85,B 0,C 180,E1 -4615.419,E2 -4615.419} C_VEL
LIN {X 0,Y 523.967,Z 216.717,A -85,B 0,C 180,E1 -4617.999,E2 -4617.999} C_VEL
LIN {X 0,Y 523.944,Z 216.719,A -85,B 0,C 180,E1 -4620.855,E2 -4620.855} C_VEL
LIN {X 0,Y 523.957,Z 216.713,A -85,B 0,C 180,E1 -4623.735,E2 -4623.735} C_VEL
LIN {X 0,Y 523.918,Z 216.725,A -85,B 0,C 180,E1 -4626.404,E2 -4626.404} C_VEL
LIN {X 0,Y 523.929,Z 216.717,A -85,B 0,C 180,E1 -4629.084,E2 -4629.084} C_VEL
LIN {X 0,Y 523.969,Z 216.703,A -85,B 0,C 180,E1 -4631.313,E2 -4631.313} C_VEL
LIN {X 0,Y 523.953,Z 216.714,A -85,B 0,C 180,E1 -4634.692,E2 -4634.692} C_VEL
LIN {X 0,Y 523.954,Z 216.721,A -85,B 0,C 180,E1 -4637.882,E2 -4637.882} C_VEL
LIN {X 0,Y 523.929,Z 216.717,A -85,B 0,C 180,E1 -4640.917,E2 -4640.917} C_VEL
LIN {X 0,Y 523.921,Z 216.726,A -85,B 0,C 180,E1 -4643.828,E2 -4643.828} C_VEL
LIN {X 0,Y 523.939,Z 216.715,A -85,B 0,C 180,E1 -4646.636,E2 -4646.636} C_VEL
LIN {X 0,Y 523.953,Z 216.718,A -85,B 0,C 180,E1 -4649.356,E2 -4649.356} C_VEL
LIN {X 0,Y 523.974,Z 216.706,A -85,B 0,C 180,E1 -4652.282,E2 -4652.282} C_VEL
LIN {X 0,Y 523.945,Z 216.714,A -85,B 0,C 180,E1 -4654.581,E2 -4654.581} C_VEL
LIN {X 0,Y 523.917,Z 216.724,A -85,B 0,C 180,E1 -4657.757,E2 -4657.757} C_VEL
LIN {X 0,Y 523.973,Z 216.704,A -85,B 0,C 180,E1 -4660.408,E2 -4660.408} C_VEL
LIN {X 0,Y 523.965,Z 216.71,A -85,B 0,C 180,E1 -4662.838,E2 -4662.838} C_VEL
LIN {X 0,Y 524.003,Z 216.713,A -85,B 0,C 180,E1 -4665.237,E2 -4665.237} C_VEL
LIN {X 0,Y 524.011,Z 216.702,A -85,B 0,C 180,E1 -4668.395,E2 -4668.395} C_VEL
LIN {X 0,Y 524.003,Z 216.711,A -85,B 0,C 180,E1 -4671.516,E2 -4671.516} C_VEL
LIN {X 0,Y 524.081,Z 216.699,A -85,B 0,C 180,E1 -4674.614,E2 -4674.614} C_VEL
LIN {X 0,Y 524.113,Z 216.692,A -85,B 0,C 180,E1 -4677.695,E2 -4677.695} C_VEL
LIN {X 0,Y 524.121,Z 216.687,A -85,B 0,C 180,E1 -4680.769,E2 -4680.769} C_VEL
LIN {X 0,Y 524.07,Z 216.705,A -85,B 0,C 180,E1 -4683.075,E2 -4683.075} C_VEL
LIN {X 0,Y 524.033,Z 216.703,A -85,B 0,C 180,E1 -4686.16,E2 -4686.16} C_VEL
LIN {X 0,Y 523.987,Z 216.706,A -85,B 0,C 180,E1 -4689.262,E2 -4689.262} C_VEL
LIN {X 0,Y 524.003,Z 216.705,A -85,B 0,C 180,E1 -4691.74,E2 -4691.74} C_VEL
LIN {X 0,Y 523.993,Z 216.714,A -85,B 0,C 180,E1 -4695.053,E2 -4695.053} C_VEL
LIN {X 0,Y 523.947,Z 216.708,A -85,B 0,C 180,E1 -4697.97,E2 -4697.97} C_VEL
LIN {X 0,Y 523.972,Z 216.71,A -85,B 0,C 180,E1 -4700.41,E2 -4700.41} C_VEL
LIN {X 0,Y 523.911,Z 216.726,A -85,B 0,C 180,E1 -4702.894,E2 -4702.894} C_VEL
LIN {X 0,Y 523.953,Z 216.711,A -85,B 0,C 180,E1 -4705.419,E2 -4705.419} C_VEL
LIN {X 0,Y 523.965,Z 216.709,A -85,B 0,C 180,E1 -4708,E2 -4708} C_VEL
LIN {X 0,Y 523.94,Z 216.721,A -85,B 0,C 180,E1 -4710.854,E2 -4710.854} C_VEL
LIN {X 0,Y 523.93,Z 216.713,A -85,B 0,C 180,E1 -4713.73,E2 -4713.73} C_VEL
LIN {X 0,Y 523.904,Z 216.727,A -85,B 0,C 180,E1 -4716.402,E2 -4716.402} C_VEL
LIN {X 0,Y 523.921,Z 216.717,A -85,B 0,C 180,E1 -4719.085,E2 -4719.085} C_VEL
LIN {X 0,Y 523.952,Z 216.719,A -85,B 0,C 180,E1 -4722.119,E2 -4722.119} C_VEL
LIN {X 0,Y 523.947,Z 216.715,A -85,B 0,C 180,E1 -4725.31,E2 -4725.31} C_VEL
LIN {X 0,Y 523.957,Z 216.71,A -85,B 0,C 180,E1 -4728.69,E2 -4728.69} C_VEL
LIN {X 0,Y 523.92,Z 216.718,A -85,B 0,C 180,E1 -4731.081,E2 -4731.081} C_VEL
LIN {X 0,Y 523.902,Z 216.725,A -85,B 0,C 180,E1 -4733.826,E2 -4733.826} C_VEL
LIN {X 0,Y 523.943,Z 216.717,A -85,B 0,C 180,E1 -4736.636,E2 -4736.636} C_VEL
LIN {X 0,Y 523.958,Z 216.718,A -85,B 0,C 180,E1 -4739.356,E2 -4739.356} C_VEL
LIN {X 0,Y 523.949,Z 216.721,A -85,B 0,C 180,E1 -4742.288,E2 -4742.288} C_VEL
LIN {X 0,Y 524.017,Z 216.902,A -85,B 0,C 180,E1 -4744.023,E2 -4744.023} C_VEL
LIN {X 0,Y 525.095,Z 223.847,A -85,B 0,C 180,E1 -4745.524,E2 -4745.524} C_VEL
LIN {X 0,Y 524.742,Z 237.102,A -85,B 0,C 180,E1 -4748.182,E2 -4748.182} C_VEL
LIN {X 0,Y 524.49,Z 249.648,A -85,B 0,C 180,E1 -4750.632,E2 -4750.632} C_VEL
LIN {X 0,Y 524.191,Z 265.228,A -85,B 0,C 180,E1 -4753.647,E2 -4753.647} C_VEL
LIN {X 0,Y 524.058,Z 271.44,A -85,B 0,C 180,E1 -4754.825,E2 -4754.825} C_VEL
LIN {X 0,Y 525.208,Z 278.564,A -85,B 0,C 180,E1 -4754.99,E2 -4754.99} C_VEL
LIN {X 0,Y 525.911,Z 284.128,A -85,B 0,C 180,E1 -4755.087,E2 -4755.087} C_VEL
LIN {X 0,Y 525.538,Z 376.329,A -85,B 0,C 180,E1 -4756.367,E2 -4756.367} C_VEL
LIN {X 0,Y 525.384,Z 386.227,A -85,B 0,C 180,E1 -4756.585,E2 -4756.585} C_VEL
LIN {X 0,Y 525.198,Z 396.205,A -85,B 0,C 180,E1 -4756.9,E2 -4756.9} C_VEL
LIN {X 0,Y 524.992,Z 406.572,A -85,B 0,C 180,E1 -4757.337,E2 -4757.337} C_VEL
LIN {X 0,Y 524.745,Z 416.651,A -85,B 0,C 180,E1 -4757.879,E2 -4757.879} C_VEL
LIN {X 0,Y 524.535,Z 426.063,A -85,B 0,C 180,E1 -4758.504,E2 -4758.504} C_VEL
LIN {X 0,Y 524.32,Z 434.577,A -85,B 0,C 180,E1 -4759.184,E2 -4759.184} C_VEL
LIN {X 0,Y 524.054,Z 442.758,A -85,B 0,C 180,E1 -4759.96,E2 -4759.96} C_VEL
LIN {X 0,Y 523.864,Z 451.315,A -85,B 0,C 180,E1 -4760.93,E2 -4760.93} C_VEL
LIN {X 0,Y 523.671,Z 459.645,A -85,B 0,C 180,E1 -4762.093,E2 -4762.093} C_VEL
LIN {X 0,Y 523.518,Z 465.3,A -85,B 0,C 180,E1 -4763.061,E2 -4763.061} C_VEL
LIN {X 0,Y 523.488,Z 470.79,A -85,B 0,C 180,E1 -4764.221,E2 -4764.221} C_VEL
LIN {X 0,Y 523.362,Z 475.108,A -85,B 0,C 180,E1 -4765.379,E2 -4765.379} C_VEL
LIN {X 0,Y 523.444,Z 477.474,A -85,B 0,C 180,E1 -4766.151,E2 -4766.151} C_VEL
LIN {X 0,Y 523.368,Z 479.267,A -85,B 0,C 180,E1 -4766.921,E2 -4766.921} C_VEL
LIN {X 0,Y 523.275,Z 481.704,A -85,B 0,C 180,E1 -4768.461,E2 -4768.461} C_VEL
LIN {X 0,Y 523.251,Z 482.29,A -85,B 0,C 180,E1 -4769.23,E2 -4769.23} C_VEL
LIN {X 0,Y 523.251,Z 482.29,A -85,B 0,C 180,E1 -4770.77,E2 -4770.77} C_VEL
LIN {X 0,Y 523.275,Z 481.704,A -85,B 0,C 180,E1 -4771.539,E2 -4771.539} C_VEL
LIN {X 0,Y 523.368,Z 479.267,A -85,B 0,C 180,E1 -4773.079,E2 -4773.079} C_VEL
LIN {X 0,Y 523.426,Z 476.325,A -85,B 0,C 180,E1 -4774.235,E2 -4774.235} C_VEL
LIN {X 0,Y 523.455,Z 472.342,A -85,B 0,C 180,E1 -4775.393,E2 -4775.393} C_VEL
LIN {X 0,Y 523.474,Z 467.31,A -85,B 0,C 180,E1 -4776.533,E2 -4776.533} C_VEL
LIN {X 0,Y 523.597,Z 461.955,A -85,B 0,C 180,E1 -4777.52,E2 -4777.52} C_VEL
LIN {X 0,Y 523.759,Z 455.639,A -85,B 0,C 180,E1 -4778.488,E2 -4778.488} C_VEL
LIN {X 0,Y 523.898,Z 449.688,A -85,B 0,C 180,E1 -4779.264,E2 -4779.264} C_VEL
LIN {X 0,Y 524.054,Z 442.758,A -85,B 0,C 180,E1 -4780.04,E2 -4780.04} C_VEL
LIN {X 0,Y 524.319,Z 434.577,A -85,B 0,C 180,E1 -4780.816,E2 -4780.816} C_VEL
LIN {X 0,Y 524.551,Z 426.063,A -85,B 0,C 180,E1 -4781.496,E2 -4781.496} C_VEL
LIN {X 0,Y 524.724,Z 417.691,A -85,B 0,C 180,E1 -4782.059,E2 -4782.059} C_VEL
LIN {X 0,Y 524.958,Z 407.579,A -85,B 0,C 180,E1 -4782.614,E2 -4782.614} C_VEL
LIN {X 0,Y 525.185,Z 398.783,A -85,B 0,C 180,E1 -4783.002,E2 -4783.002} C_VEL
LIN {X 0,Y 525.352,Z 388.851,A -85,B 0,C 180,E1 -4783.342,E2 -4783.342} C_VEL
LIN {X 0,Y 525.5,Z 378.993,A -85,B 0,C 180,E1 -4783.584,E2 -4783.584} C_VEL
LIN {X 0,Y 525.67,Z 354.382,A -85,B 0,C 180,E1 -4783.95,E2 -4783.95} C_VEL
LIN {X 0,Y 525.765,Z 281.83,A -85,B 0,C 180,E1 -4784.949,E2 -4784.949} C_VEL
LIN {X 0,Y 524.098,Z 271.653,A -85,B 0,C 180,E1 -4785.158,E2 -4785.158} C_VEL
LIN {X 0,Y 524.057,Z 269.351,A -85,B 0,C 180,E1 -4785.558,E2 -4785.558} C_VEL
LIN {X 0,Y 524.421,Z 254.874,A -85,B 0,C 180,E1 -4788.357,E2 -4788.357} C_VEL
LIN {X 0,Y 524.706,Z 240.234,A -85,B 0,C 180,E1 -4791.201,E2 -4791.201} C_VEL
LIN {X 0,Y 525.101,Z 225.824,A -85,B 0,C 180,E1 -4794.075,E2 -4794.075} C_VEL
LIN {X 0,Y 524.657,Z 220.582,A -85,B 0,C 180,E1 -4795.17,E2 -4795.17} C_VEL
LIN {X 0,Y 523.969,Z 216.748,A -85,B 0,C 180,E1 -4796.042,E2 -4796.042} C_VEL
LIN {X 0,Y 523.93,Z 216.721,A -85,B 0,C 180,E1 -4798.875,E2 -4798.875} C_VEL
LIN {X 0,Y 523.923,Z 216.724,A -85,B 0,C 180,E1 -4801.544,E2 -4801.544} C_VEL
LIN {X 0,Y 523.934,Z 216.72,A -85,B 0,C 180,E1 -4804.29,E2 -4804.29} C_VEL
LIN {X 0,Y 523.909,Z 216.72,A -85,B 0,C 180,E1 -4807.132,E2 -4807.132} C_VEL
LIN {X 0,Y 523.939,Z 216.714,A -85,B 0,C 180,E1 -4810.129,E2 -4810.129} C_VEL
LIN {X 0,Y 523.923,Z 216.72,A -85,B 0,C 180,E1 -4813.166,E2 -4813.166} C_VEL
LIN {X 0,Y 523.938,Z 216.722,A -85,B 0,C 180,E1 -4815.771,E2 -4815.771} C_VEL
LIN {X 0,Y 523.94,Z 216.716,A -85,B 0,C 180,E1 -4818.907,E2 -4818.907} C_VEL
LIN {X 0,Y 523.916,Z 216.723,A -85,B 0,C 180,E1 -4821.898,E2 -4821.898} C_VEL
LIN {X 0,Y 523.924,Z 216.717,A -85,B 0,C 180,E1 -4824.911,E2 -4824.911} C_VEL
LIN {X 0,Y 523.935,Z 216.722,A -85,B 0,C 180,E1 -4827.679,E2 -4827.679} C_VEL
LIN {X 0,Y 523.954,Z 216.714,A -85,B 0,C 180,E1 -4830.676,E2 -4830.676} C_VEL
LIN {X 0,Y 523.974,Z 216.711,A -85,B 0,C 180,E1 -4833.728,E2 -4833.728} C_VEL
LIN {X 0,Y 523.926,Z 216.717,A -85,B 0,C 180,E1 -4836.27,E2 -4836.27} C_VEL
LIN {X 0,Y 523.946,Z 216.717,A -85,B 0,C 180,E1 -4838.766,E2 -4838.766} C_VEL
LIN {X 0,Y 523.947,Z 216.713,A -85,B 0,C 180,E1 -4841.22,E2 -4841.22} C_VEL
LIN {X 0,Y 523.929,Z 216.718,A -85,B 0,C 180,E1 -4843.638,E2 -4843.638} C_VEL
LIN {X 0,Y 523.938,Z 216.715,A -85,B 0,C 180,E1 -4846.028,E2 -4846.028} C_VEL
LIN {X 0,Y 524.013,Z 216.705,A -85,B 0,C 180,E1 -4848.394,E2 -4848.394} C_VEL
LIN {X 0,Y 523.988,Z 216.707,A -85,B 0,C 180,E1 -4851.515,E2 -4851.515} C_VEL
LIN {X 0,Y 524.08,Z 216.702,A -85,B 0,C 180,E1 -4854.613,E2 -4854.613} C_VEL
LIN {X 0,Y 524.112,Z 216.692,A -85,B 0,C 180,E1 -4857.694,E2 -4857.694} C_VEL
LIN {X 0,Y 524.123,Z 216.691,A -85,B 0,C 180,E1 -4860.768,E2 -4860.768} C_VEL
LIN {X 0,Y 524.069,Z 216.703,A -85,B 0,C 180,E1 -4863.074,E2 -4863.074} C_VEL
LIN {X 0,Y 524.037,Z 216.706,A -85,B 0,C 180,E1 -4866.159,E2 -4866.159} C_VEL
LIN {X 0,Y 524.003,Z 216.711,A -85,B 0,C 180,E1 -4868.484,E2 -4868.484} C_VEL
LIN {X 0,Y 524.001,Z 216.704,A -85,B 0,C 180,E1 -4871.739,E2 -4871.739} C_VEL
LIN {X 0,Y 523.992,Z 216.711,A -85,B 0,C 180,E1 -4875.052,E2 -4875.052} C_VEL
LIN {X 0,Y 523.962,Z 216.712,A -85,B 0,C 180,E1 -4877.969,E2 -4877.969} C_VEL
LIN {X 0,Y 523.97,Z 216.714,A -85,B 0,C 180,E1 -4880.41,E2 -4880.41} C_VEL
LIN {X 0,Y 523.908,Z 216.722,A -85,B 0,C 180,E1 -4882.893,E2 -4882.893} C_VEL
LIN {X 0,Y 523.982,Z 216.714,A -85,B 0,C 180,E1 -4886.019,E2 -4886.019} C_VEL
LIN {X 0,Y 523.936,Z 216.716,A -85,B 0,C 180,E1 -4888.874,E2 -4888.874} C_VEL
LIN {X 0,Y 523.921,Z 216.72,A -85,B 0,C 180,E1 -4891.544,E2 -4891.544} C_VEL
LIN {X 0,Y 523.938,Z 216.718,A -85,B 0,C 180,E1 -4894.289,E2 -4894.289} C_VEL
LIN {X 0,Y 523.908,Z 216.72,A -85,B 0,C 180,E1 -4897.132,E2 -4897.132} C_VEL
LIN {X 0,Y 523.934,Z 216.719,A -85,B 0,C 180,E1 -4900.13,E2 -4900.13} C_VEL
LIN {X 0,Y 523.937,Z 216.719,A -85,B 0,C 180,E1 -4902.459,E2 -4902.459} C_VEL
LIN {X 0,Y 523.953,Z 216.714,A -85,B 0,C 180,E1 -4905.308,E2 -4905.308} C_VEL
LIN {X 0,Y 523.916,Z 216.71,A -85,B 0,C 180,E1 -4906.913,E2 -4906.913} C_VEL
LIN {X 0,Y 523.254,Z 216.796,A -85,B 0,C 180,E1 -4907.554,E2 -4907.554} C_VEL
LIN {X 0,Y 520.426,Z 217.155,A -85,B 0,C 180,E1 -4908.596,E2 -4908.596} C_VEL
LIN {X 0,Y 518.028,Z 217.457,A -85,B 0,C 180,E1 -4909.436,E2 -4909.436} C_VEL
LIN {X 0,Y 516.989,Z 217.586,A -85,B 0,C 180,E1 -4910.083,E2 -4910.083} C_VEL
LIN {X 0,Y 516.899,Z 217.595,A -85,B 0,C 180,E1 -4910.303,E2 -4910.303} C_VEL
LIN {X 0,Y 516.881,Z 217.599,A -85,B 0,C 180,E1 -4913.342,E2 -4913.342} C_VEL
LIN {X 0,Y 516.907,Z 217.593,A -85,B 0,C 180,E1 -4916.121,E2 -4916.121} C_VEL
LIN {X 0,Y 516.889,Z 217.596,A -85,B 0,C 180,E1 -4918.935,E2 -4918.935} C_VEL
LIN {X 0,Y 516.916,Z 217.593,A -85,B 0,C 180,E1 -4921.585,E2 -4921.585} C_VEL
LIN {X 0,Y 516.928,Z 217.592,A -85,B 0,C 180,E1 -4924.211,E2 -4924.211} C_VEL
LIN {X 0,Y 516.862,Z 217.6,A -85,B 0,C 180,E1 -4926.776,E2 -4926.776} C_VEL
LIN {X 0,Y 516.936,Z 217.595,A -85,B 0,C 180,E1 -4929.731,E2 -4929.731} C_VEL
LIN {X 0,Y 516.926,Z 217.592,A -85,B 0,C 180,E1 -4932.596,E2 -4932.596} C_VEL
LIN {X 0,Y 516.948,Z 217.594,A -85,B 0,C 180,E1 -4935.03,E2 -4935.03} C_VEL
LIN {X 0,Y 516.962,Z 217.588,A -85,B 0,C 180,E1 -4938.234,E2 -4938.234} C_VEL
LIN {X 0,Y 516.967,Z 217.592,A -85,B 0,C 180,E1 -4941.4,E2 -4941.4} C_VEL
LIN {X 0,Y 517.014,Z 217.582,A -85,B 0,C 180,E1 -4943.757,E2 -4943.757} C_VEL
LIN {X 0,Y 517.083,Z 217.574,A -85,B 0,C 180,E1 -4947.663,E2 -4947.663} C_VEL
LIN {X 0,Y 517.091,Z 217.577,A -85,B 0,C 180,E1 -4950.779,E2 -4950.779} C_VEL
LIN {X 0,Y 517.01,Z 217.587,A -85,B 0,C 180,E1 -4953.117,E2 -4953.117} C_VEL
LIN {X 0,Y 517.014,Z 217.582,A -85,B 0,C 180,E1 -4956.243,E2 -4956.243} C_VEL
LIN {X 0,Y 516.951,Z 217.59,A -85,B 0,C 180,E1 -4959.389,E2 -4959.389} C_VEL
LIN {X 0,Y 516.949,Z 217.589,A -85,B 0,C 180,E1 -4961.808,E2 -4961.808} C_VEL
LIN {X 0,Y 516.944,Z 217.593,A -85,B 0,C 180,E1 -4965.148,E2 -4965.148} C_VEL
LIN {X 0,Y 516.922,Z 217.595,A -85,B 0,C 180,E1 -4968.222,E2 -4968.222} C_VEL
LIN {X 0,Y 516.909,Z 217.6,A -85,B 0,C 180,E1 -4970.702,E2 -4970.702} C_VEL
LIN {X 0,Y 516.9,Z 217.597,A -85,B 0,C 180,E1 -4974.072,E2 -4974.072} C_VEL
LIN {X 0,Y 516.923,Z 217.597,A -85,B 0,C 180,E1 -4976.658,E2 -4976.658} C_VEL
LIN {X 0,Y 516.908,Z 217.585,A -85,B 0,C 180,E1 -4979.524,E2 -4979.524} C_VEL
LIN {X 0,Y 516.897,Z 217.597,A -85,B 0,C 180,E1 -4982.544,E2 -4982.544} C_VEL
LIN {X 0,Y 516.875,Z 217.59,A -85,B 0,C 180,E1 -4985.332,E2 -4985.332} C_VEL
LIN {X 0,Y 516.879,Z 217.601,A -85,B 0,C 180,E1 -4987.944,E2 -4987.944} C_VEL
LIN {X 0,Y 516.901,Z 217.585,A -85,B 0,C 180,E1 -4990.74,E2 -4990.74} C_VEL
LIN {X 0,Y 516.879,Z 217.592,A -85,B 0,C 180,E1 -4993.903,E2 -4993.903} C_VEL
LIN {X 0,Y 516.879,Z 217.604,A -85,B 0,C 180,E1 -4996.107,E2 -4996.107} C_VEL
LIN {X 0,Y 516.892,Z 217.59,A -85,B 0,C 180,E1 -4999.26,E2 -4999.26} C_VEL
LIN {X 0,Y 516.862,Z 217.602,A -85,B 0,C 180,E1 -5002.275,E2 -5002.275} C_VEL
LIN {X 0,Y 516.889,Z 217.591,A -85,B 0,C 180,E1 -5005.176,E2 -5005.176} C_VEL
LIN {X 0,Y 516.874,Z 217.604,A -85,B 0,C 180,E1 -5007.976,E2 -5007.976} C_VEL
LIN {X 0,Y 516.919,Z 217.589,A -85,B 0,C 180,E1 -5010.696,E2 -5010.696} C_VEL
LIN {X 0,Y 516.94,Z 217.591,A -85,B 0,C 180,E1 -5013.804,E2 -5013.804} C_VEL
LIN {X 0,Y 516.863,Z 217.598,A -85,B 0,C 180,E1 -5016.777,E2 -5016.777} C_VEL
LIN {X 0,Y 516.937,Z 217.586,A -85,B 0,C 180,E1 -5019.732,E2 -5019.732} C_VEL
LIN {X 0,Y 516.927,Z 217.585,A -85,B 0,C 180,E1 -5022.597,E2 -5022.597} C_VEL
LIN {X 0,Y 516.949,Z 217.589,A -85,B 0,C 180,E1 -5025.031,E2 -5025.031} C_VEL
LIN {X 0,Y 516.964,Z 217.58,A -85,B 0,C 180,E1 -5028.234,E2 -5028.234} C_VEL
LIN {X 0,Y 516.968,Z 217.584,A -85,B 0,C 180,E1 -5031.4,E2 -5031.4} C_VEL
LIN {X 0,Y 517.002,Z 217.583,A -85,B 0,C 180,E1 -5033.757,E2 -5033.757} C_VEL
LIN {X 0,Y 517.01,Z 217.582,A -85,B 0,C 180,E1 -5036.883,E2 -5036.883} C_VEL
LIN {X 0,Y 517.085,Z 217.56,A -85,B 0,C 180,E1 -5040,E2 -5040} C_VEL
LIN {X 0,Y 517.012,Z 217.585,A -85,B 0,C 180,E1 -5043.117,E2 -5043.117} C_VEL
LIN {X 0,Y 516.994,Z 217.58,A -85,B 0,C 180,E1 -5046.244,E2 -5046.244} C_VEL
LIN {X 0,Y 516.943,Z 217.581,A -85,B 0,C 180,E1 -5049.39,E2 -5049.39} C_VEL
LIN {X 0,Y 516.952,Z 217.583,A -85,B 0,C 180,E1 -5051.807,E2 -5051.807} C_VEL
LIN {X 0,Y 516.945,Z 217.59,A -85,B 0,C 180,E1 -5055.147,E2 -5055.147} C_VEL
LIN {X 0,Y 516.916,Z 217.585,A -85,B 0,C 180,E1 -5058.223,E2 -5058.223} C_VEL
LIN {X 0,Y 516.912,Z 217.593,A -85,B 0,C 180,E1 -5060.702,E2 -5060.702} C_VEL
LIN {X 0,Y 516.903,Z 217.593,A -85,B 0,C 180,E1 -5064.073,E2 -5064.073} C_VEL
LIN {X 0,Y 516.925,Z 217.59,A -85,B 0,C 180,E1 -5066.658,E2 -5066.658} C_VEL
LIN {X 0,Y 516.91,Z 217.591,A -85,B 0,C 180,E1 -5069.524,E2 -5069.524} C_VEL
LIN {X 0,Y 516.895,Z 217.598,A -85,B 0,C 180,E1 -5072.543,E2 -5072.543} C_VEL
LIN {X 0,Y 516.866,Z 217.595,A -85,B 0,C 180,E1 -5075.33,E2 -5075.33} C_VEL
LIN {X 0,Y 516.881,Z 217.598,A -85,B 0,C 180,E1 -5077.943,E2 -5077.943} C_VEL
LIN {X 0,Y 516.884,Z 217.598,A -85,B 0,C 180,E1 -5080.742,E2 -5080.742} C_VEL
LIN {X 0,Y 516.885,Z 217.597,A -85,B 0,C 180,E1 -5082.832,E2 -5082.832} C_VEL
LIN {X 0,Y 516.884,Z 217.601,A -85,B 0,C 180,E1 -5086.097,E2 -5086.097} C_VEL
LIN {X 0,Y 516.915,Z 217.591,A -85,B 0,C 180,E1 -5088.399,E2 -5088.399} C_VEL
LIN {X 0,Y 516.883,Z 217.595,A -85,B 0,C 180,E1 -5091.285,E2 -5091.285} C_VEL
LIN {X 0,Y 516.873,Z 217.599,A -85,B 0,C 180,E1 -5094.22,E2 -5094.22} C_VEL
LIN {X 0,Y 516.897,Z 217.593,A -85,B 0,C 180,E1 -5097.053,E2 -5097.053} C_VEL
LIN {X 0,Y 516.894,Z 217.601,A -85,B 0,C 180,E1 -5099.797,E2 -5099.797} C_VEL
LIN {X 0,Y 516.902,Z 217.599,A -85,B 0,C 180,E1 -5102.466,E2 -5102.466} C_VEL
LIN {X 0,Y 516.978,Z 217.771,A -85,B 0,C 180,E1 -5103.846,E2 -5103.846} C_VEL
LIN {X 0,Y 518.098,Z 224.579,A -85,B 0,C 180,E1 -5105.348,E2 -5105.348} C_VEL
LIN {X 0,Y 517.895,Z 234.308,A -85,B 0,C 180,E1 -5107.337,E2 -5107.337} C_VEL
LIN {X 0,Y 517.602,Z 246.885,A -85,B 0,C 180,E1 -5109.843,E2 -5109.843} C_VEL
LIN {X 0,Y 517.255,Z 260.936,A -85,B 0,C 180,E1 -5112.608,E2 -5112.608} C_VEL
LIN {X 0,Y 517.046,Z 271.271,A -85,B 0,C 180,E1 -5114.617,E2 -5114.617} C_VEL
LIN {X 0,Y 518.36,Z 279.509,A -85,B 0,C 180,E1 -5114.803,E2 -5114.803} C_VEL
LIN {X 0,Y 519.058,Z 284.808,A -85,B 0,C 180,E1 -5114.898,E2 -5114.898} C_VEL
LIN {X 0,Y 518.651,Z 376.137,A -85,B 0,C 180,E1 -5116.183,E2 -5116.183} C_VEL
LIN {X 0,Y 518.495,Z 386.035,A -85,B 0,C 180,E1 -5116.403,E2 -5116.403} C_VEL
LIN {X 0,Y 518.273,Z 396.012,A -85,B 0,C 180,E1 -5116.722,E2 -5116.722} C_VEL
LIN {X 0,Y 518.054,Z 406.379,A -85,B 0,C 180,E1 -5117.165,E2 -5117.165} C_VEL
LIN {X 0,Y 517.791,Z 416.084,A -85,B 0,C 180,E1 -5117.691,E2 -5117.691} C_VEL
LIN {X 0,Y 517.568,Z 424.516,A -85,B 0,C 180,E1 -5118.248,E2 -5118.248} C_VEL
LIN {X 0,Y 517.341,Z 433.248,A -85,B 0,C 180,E1 -5118.937,E2 -5118.937} C_VEL
LIN {X 0,Y 517.061,Z 440.644,A -85,B 0,C 180,E1 -5119.625,E2 -5119.625} C_VEL
LIN {X 0,Y 516.921,Z 447.867,A -85,B 0,C 180,E1 -5120.413,E2 -5120.413} C_VEL
LIN {X 0,Y 516.72,Z 454.069,A -85,B 0,C 180,E1 -5121.198,E2 -5121.198} C_VEL
LIN {X 0,Y 516.56,Z 460.606,A -85,B 0,C 180,E1 -5122.18,E2 -5122.18} C_VEL
LIN {X 0,Y 516.444,Z 465.107,A -85,B 0,C 180,E1 -5122.965,E2 -5122.965} C_VEL
LIN {X 0,Y 516.402,Z 470.596,A -85,B 0,C 180,E1 -5124.142,E2 -5124.142} C_VEL
LIN {X 0,Y 516.273,Z 474.915,A -85,B 0,C 180,E1 -5125.315,E2 -5125.315} C_VEL
LIN {X 0,Y 516.353,Z 477.281,A -85,B 0,C 180,E1 -5126.098,E2 -5126.098} C_VEL
LIN {X 0,Y 516.283,Z 479.074,A -85,B 0,C 180,E1 -5126.879,E2 -5126.879} C_VEL
LIN {X 0,Y 516.192,Z 481.512,A -85,B 0,C 180,E1 -5128.44,E2 -5128.44} C_VEL
LIN {X 0,Y 516.161,Z 482.098,A -85,B 0,C 180,E1 -5129.22,E2 -5129.22} C_VEL
LIN {X 0,Y 516.161,Z 482.098,A -85,B 0,C 180,E1 -5130.78,E2 -5130.78} C_VEL
LIN {X 0,Y 516.192,Z 481.512,A -85,B 0,C 180,E1 -5131.56,E2 -5131.56} C_VEL
LIN {X 0,Y 516.283,Z 479.074,A -85,B 0,C 180,E1 -5133.121,E2 -5133.121} C_VEL
LIN {X 0,Y 516.314,Z 476.131,A -85,B 0,C 180,E1 -5134.293,E2 -5134.293} C_VEL
LIN {X 0,Y 516.367,Z 472.149,A -85,B 0,C 180,E1 -5135.467,E2 -5135.467} C_VEL
LIN {X 0,Y 516.389,Z 466.961,A -85,B 0,C 180,E1 -5136.655,E2 -5136.655} C_VEL
LIN {X 0,Y 516.537,Z 461.762,A -85,B 0,C 180,E1 -5137.623,E2 -5137.623} C_VEL
LIN {X 0,Y 516.714,Z 455.446,A -85,B 0,C 180,E1 -5138.605,E2 -5138.605} C_VEL
LIN {X 0,Y 516.875,Z 449.494,A -85,B 0,C 180,E1 -5139.391,E2 -5139.391} C_VEL
LIN {X 0,Y 517.015,Z 442.564,A -85,B 0,C 180,E1 -5140.178,E2 -5140.178} C_VEL
LIN {X 0,Y 517.312,Z 434.384,A -85,B 0,C 180,E1 -5140.964,E2 -5140.964} C_VEL
LIN {X 0,Y 517.568,Z 425.87,A -85,B 0,C 180,E1 -5141.653,E2 -5141.653} C_VEL
LIN {X 0,Y 517.768,Z 417.404,A -85,B 0,C 180,E1 -5142.229,E2 -5142.229} C_VEL
LIN {X 0,Y 518.039,Z 407.387,A -85,B 0,C 180,E1 -5142.786,E2 -5142.786} C_VEL
LIN {X 0,Y 518.239,Z 398.589,A -85,B 0,C 180,E1 -5143.179,E2 -5143.179} C_VEL
LIN {X 0,Y 518.457,Z 388.658,A -85,B 0,C 180,E1 -5143.523,E2 -5143.523} C_VEL
LIN {X 0,Y 518.598,Z 378.8,A -85,B 0,C 180,E1 -5143.769,E2 -5143.769} C_VEL
LIN {X 0,Y 518.781,Z 354.189,A -85,B 0,C 180,E1 -5144.139,E2 -5144.139} C_VEL
LIN {X 0,Y 518.884,Z 282.306,A -85,B 0,C 180,E1 -5145.142,E2 -5145.142} C_VEL
LIN {X 0,Y 517.056,Z 271.449,A -85,B 0,C 180,E1 -5145.37,E2 -5145.37} C_VEL
LIN {X 0,Y 517.038,Z 269.17,A -85,B 0,C 180,E1 -5145.775,E2 -5145.775} C_VEL
LIN {X 0,Y 517.399,Z 254.742,A -85,B 0,C 180,E1 -5148.615,E2 -5148.615} C_VEL
LIN {X 0,Y 517.711,Z 241.146,A -85,B 0,C 180,E1 -5151.293,E2 -5151.293} C_VEL
LIN {X 0,Y 518.141,Z 227.69,A -85,B 0,C 180,E1 -5154.011,E2 -5154.011} C_VEL
LIN {X 0,Y 517.822,Z 222.538,A -85,B 0,C 180,E1 -5155.096,E2 -5155.096} C_VEL
LIN {X 0,Y 516.935,Z 217.63,A -85,B 0,C 180,E1 -5156.22,E2 -5156.22} C_VEL
LIN {X 0,Y 516.913,Z 217.597,A -85,B 0,C 180,E1 -5159.523,E2 -5159.523} C_VEL
LIN {X 0,Y 516.898,Z 217.595,A -85,B 0,C 180,E1 -5162.543,E2 -5162.543} C_VEL
LIN {X 0,Y 516.868,Z 217.598,A -85,B 0,C 180,E1 -5165.329,E2 -5165.329} C_VEL
LIN {X 0,Y 516.882,Z 217.602,A -85,B 0,C 180,E1 -5167.943,E2 -5167.943} C_VEL
LIN {X 0,Y 516.884,Z 217.588,A -85,B 0,C 180,E1 -5170.741,E2 -5170.741} C_VEL
LIN {X 0,Y 516.885,Z 217.595,A -85,B 0,C 180,E1 -5172.831,E2 -5172.831} C_VEL
LIN {X 0,Y 516.884,Z 217.598,A -85,B 0,C 180,E1 -5176.097,E2 -5176.097} C_VEL
LIN {X 0,Y 516.914,Z 217.591,A -85,B 0,C 180,E1 -5178.398,E2 -5178.398} C_VEL
LIN {X 0,Y 516.881,Z 217.597,A -85,B 0,C 180,E1 -5181.284,E2 -5181.284} C_VEL
LIN {X 0,Y 516.871,Z 217.595,A -85,B 0,C 180,E1 -5184.219,E2 -5184.219} C_VEL
LIN {X 0,Y 516.881,Z 217.594,A -85,B 0,C 180,E1 -5187.052,E2 -5187.052} C_VEL
LIN {X 0,Y 516.887,Z 217.597,A -85,B 0,C 180,E1 -5189.796,E2 -5189.796} C_VEL
LIN {X 0,Y 516.926,Z 217.584,A -85,B 0,C 180,E1 -5192.467,E2 -5192.467} C_VEL
LIN {X 0,Y 516.909,Z 217.593,A -85,B 0,C 180,E1 -5195.071,E2 -5195.071} C_VEL
LIN {X 0,Y 516.885,Z 217.594,A -85,B 0,C 180,E1 -5198.462,E2 -5198.462} C_VEL
LIN {X 0,Y 516.9,Z 217.592,A -85,B 0,C 180,E1 -5200.954,E2 -5200.954} C_VEL
LIN {X 0,Y 516.905,Z 217.595,A -85,B 0,C 180,E1 -5203.41,E2 -5203.41} C_VEL
LIN {X 0,Y 516.894,Z 217.594,A -85,B 0,C 180,E1 -5205.833,E2 -5205.833} C_VEL
LIN {X 0,Y 516.966,Z 217.582,A -85,B 0,C 180,E1 -5208.233,E2 -5208.233} C_VEL
LIN {X 0,Y 516.956,Z 217.583,A -85,B 0,C 180,E1 -5211.399,E2 -5211.399} C_VEL
LIN {X 0,Y 517.026,Z 217.58,A -85,B 0,C 180,E1 -5214.54,E2 -5214.54} C_VEL
LIN {X 0,Y 517.084,Z 217.567,A -85,B 0,C 180,E1 -5217.663,E2 -5217.663} C_VEL
LIN {X 0,Y 517.093,Z 217.565,A -85,B 0,C 180,E1 -5220.778,E2 -5220.778} C_VEL
LIN {X 0,Y 517.01,Z 217.582,A -85,B 0,C 180,E1 -5223.117,E2 -5223.117} C_VEL
LIN {X 0,Y 517.002,Z 217.583,A -85,B 0,C 180,E1 -5226.243,E2 -5226.243} C_VEL
LIN {X 0,Y 516.952,Z 217.577,A -85,B 0,C 180,E1 -5229.389,E2 -5229.389} C_VEL
LIN {X 0,Y 516.951,Z 217.582,A -85,B 0,C 180,E1 -5231.807,E2 -5231.807} C_VEL
LIN {X 0,Y 516.945,Z 217.588,A -85,B 0,C 180,E1 -5235.147,E2 -5235.147} C_VEL
LIN {X 0,Y 516.923,Z 217.592,A -85,B 0,C 180,E1 -5238.222,E2 -5238.222} C_VEL
LIN {X 0,Y 516.91,Z 217.594,A -85,B 0,C 180,E1 -5240.701,E2 -5240.701} C_VEL
LIN {X 0,Y 516.888,Z 217.6,A -85,B 0,C 180,E1 -5244.073,E2 -5244.073} C_VEL
LIN {X 0,Y 516.922,Z 217.585,A -85,B 0,C 180,E1 -5246.657,E2 -5246.657} C_VEL
LIN {X 0,Y 516.908,Z 217.591,A -85,B 0,C 180,E1 -5249.523,E2 -5249.523} C_VEL
LIN {X 0,Y 516.895,Z 217.595,A -85,B 0,C 180,E1 -5252.543,E2 -5252.543} C_VEL
LIN {X 0,Y 516.876,Z 217.592,A -85,B 0,C 180,E1 -5255.331,E2 -5255.331} C_VEL
LIN {X 0,Y 516.879,Z 217.604,A -85,B 0,C 180,E1 -5257.943,E2 -5257.943} C_VEL
LIN {X 0,Y 516.882,Z 217.592,A -85,B 0,C 180,E1 -5260.741,E2 -5260.741} C_VEL
LIN {X 0,Y 516.901,Z 217.593,A -85,B 0,C 180,E1 -5262.829,E2 -5262.829} C_VEL
LIN {X 0,Y 516.919,Z 217.589,A -85,B 0,C 180,E1 -5265.01,E2 -5265.01} C_VEL
LIN {X 0,Y 516.919,Z 217.583,A -85,B 0,C 180,E1 -5268.397,E2 -5268.397} C_VEL
LIN {X 0,Y 516.899,Z 217.595,A -85,B 0,C 180,E1 -5270.303,E2 -5270.303} C_VEL
LIN {X 0,Y 516.218,Z 217.678,A -85,B 0,C 180,E1 -5270.953,E2 -5270.953} C_VEL
LIN {X 0,Y 513.365,Z 218.04,A -85,B 0,C 180,E1 -5272.008,E2 -5272.008} C_VEL
LIN {X 0,Y 510.956,Z 218.344,A -85,B 0,C 180,E1 -5272.858,E2 -5272.858} C_VEL
LIN {X 0,Y 509.916,Z 218.469,A -85,B 0,C 180,E1 -5273.514,E2 -5273.514} C_VEL
LIN {X 0,Y 509.827,Z 218.476,A -85,B 0,C 180,E1 -5273.737,E2 -5273.737} C_VEL
LIN {X 0,Y 509.858,Z 218.468,A -85,B 0,C 180,E1 -5276.539,E2 -5276.539} C_VEL
LIN {X 0,Y 509.843,Z 218.478,A -85,B 0,C 180,E1 -5279.334,E2 -5279.334} C_VEL
LIN {X 0,Y 509.891,Z 218.47,A -85,B 0,C 180,E1 -5282.055,E2 -5282.055} C_VEL
LIN {X 0,Y 509.873,Z 218.47,A -85,B 0,C 180,E1 -5284.704,E2 -5284.704} C_VEL
LIN {X 0,Y 509.823,Z 218.483,A -85,B 0,C 180,E1 -5287.458,E2 -5287.458} C_VEL
LIN {X 0,Y 509.913,Z 218.468,A -85,B 0,C 180,E1 -5289.845,E2 -5289.845} C_VEL
LIN {X 0,Y 509.881,Z 218.475,A -85,B 0,C 180,E1 -5293.175,E2 -5293.175} C_VEL
LIN {X 0,Y 509.87,Z 218.475,A -85,B 0,C 180,E1 -5295.634,E2 -5295.634} C_VEL
LIN {X 0,Y 509.911,Z 218.47,A -85,B 0,C 180,E1 -5298.875,E2 -5298.875} C_VEL
LIN {X 0,Y 509.948,Z 218.462,A -85,B 0,C 180,E1 -5302.078,E2 -5302.078} C_VEL
LIN {X 0,Y 509.983,Z 218.458,A -85,B 0,C 180,E1 -5304.464,E2 -5304.464} C_VEL
LIN {X 0,Y 510.054,Z 218.45,A -85,B 0,C 180,E1 -5307.631,E2 -5307.631} C_VEL
LIN {X 0,Y 510.061,Z 218.452,A -85,B 0,C 180,E1 -5310.789,E2 -5310.789} C_VEL
LIN {X 0,Y 509.952,Z 218.466,A -85,B 0,C 180,E1 -5313.16,E2 -5313.16} C_VEL
LIN {X 0,Y 509.981,Z 218.459,A -85,B 0,C 180,E1 -5316.33,E2 -5316.33} C_VEL
LIN {X 0,Y 509.913,Z 218.472,A -85,B 0,C 180,E1 -5318.72,E2 -5318.72} C_VEL
LIN {X 0,Y 509.901,Z 218.468,A -85,B 0,C 180,E1 -5321.932,E2 -5321.932} C_VEL
LIN {X 0,Y 509.89,Z 218.47,A -85,B 0,C 180,E1 -5325.242,E2 -5325.242} C_VEL
LIN {X 0,Y 509.885,Z 218.47,A -85,B 0,C 180,E1 -5328.001,E2 -5328.001} C_VEL
LIN {X 0,Y 509.847,Z 218.476,A -85,B 0,C 180,E1 -5331.002,E2 -5331.002} C_VEL
LIN {X 0,Y 509.861,Z 218.478,A -85,B 0,C 180,E1 -5334.426,E2 -5334.426} C_VEL
LIN {X 0,Y 509.882,Z 218.47,A -85,B 0,C 180,E1 -5337.056,E2 -5337.056} C_VEL
LIN {X 0,Y 509.854,Z 218.464,A -85,B 0,C 180,E1 -5339.751,E2 -5339.751} C_VEL
LIN {X 0,Y 509.873,Z 218.469,A -85,B 0,C 180,E1 -5342.775,E2 -5342.775} C_VEL
LIN {X 0,Y 509.836,Z 218.467,A -85,B 0,C 180,E1 -5345.581,E2 -5345.581} C_VEL
LIN {X 0,Y 509.849,Z 218.478,A -85,B 0,C 180,E1 -5348.338,E2 -5348.338} C_VEL
LIN {X 0,Y 509.862,Z 218.46,A -85,B 0,C 180,E1 -5351.425,E2 -5351.425} C_VEL
LIN {X 0,Y 509.853,Z 218.471,A -85,B 0,C 180,E1 -5354.668,E2 -5354.668} C_VEL
LIN {X 0,Y 509.876,Z 218.472,A -85,B 0,C 180,E1 -5358.101,E2 -5358.101} C_VEL
LIN {X 0,Y 509.853,Z 218.471,A -85,B 0,C 180,E1 -5360.649,E2 -5360.649} C_VEL
LIN {X 0,Y 509.831,Z 218.479,A -85,B 0,C 180,E1 -5363.648,E2 -5363.648} C_VEL
LIN {X 0,Y 509.858,Z 218.469,A -85,B 0,C 180,E1 -5366.54,E2 -5366.54} C_VEL
LIN {X 0,Y 509.843,Z 218.475,A -85,B 0,C 180,E1 -5369.335,E2 -5369.335} C_VEL
LIN {X 0,Y 509.889,Z 218.462,A -85,B 0,C 180,E1 -5372.055,E2 -5372.055} C_VEL
LIN {X 0,Y 509.838,Z 218.471,A -85,B 0,C 180,E1 -5374.702,E2 -5374.702} C_VEL
LIN {X 0,Y 509.825,Z 218.481,A -85,B 0,C 180,E1 -5377.458,E2 -5377.458} C_VEL
LIN {X 0,Y 509.915,Z 218.459,A -85,B 0,C 180,E1 -5379.845,E2 -5379.845} C_VEL
LIN {X 0,Y 509.883,Z 218.467,A -85,B 0,C 180,E1 -5383.175,E2 -5383.175} C_VEL
LIN {X 0,Y 509.872,Z 218.475,A -85,B 0,C 180,E1 -5385.635,E2 -5385.635} C_VEL
LIN {X 0,Y 509.912,Z 218.46,A -85,B 0,C 180,E1 -5388.875,E2 -5388.875} C_VEL
LIN {X 0,Y 509.95,Z 218.456,A -85,B 0,C 180,E1 -5392.079,E2 -5392.079} C_VEL
LIN {X 0,Y 509.979,Z 218.455,A -85,B 0,C 180,E1 -5394.465,E2 -5394.465} C_VEL
LIN {X 0,Y 510.055,Z 218.443,A -85,B 0,C 180,E1 -5397.631,E2 -5397.631} C_VEL
LIN {X 0,Y 510.062,Z 218.437,A -85,B 0,C 180,E1 -5400.79,E2 -5400.79} C_VEL
LIN {X 0,Y 509.954,Z 218.465,A -85,B 0,C 180,E1 -5403.161,E2 -5403.161} C_VEL
LIN {X 0,Y 509.941,Z 218.459,A -85,B 0,C 180,E1 -5406.33,E2 -5406.33} C_VEL
LIN {X 0,Y 509.904,Z 218.463,A -85,B 0,C 180,E1 -5408.721,E2 -5408.721} C_VEL
LIN {X 0,Y 509.904,Z 218.461,A -85,B 0,C 180,E1 -5411.932,E2 -5411.932} C_VEL
LIN {X 0,Y 509.894,Z 218.467,A -85,B 0,C 180,E1 -5415.242,E2 -5415.242} C_VEL
LIN {X 0,Y 509.861,Z 218.465,A -85,B 0,C 180,E1 -5418.484,E2 -5418.484} C_VEL
LIN {X 0,Y 509.85,Z 218.475,A -85,B 0,C 180,E1 -5421.002,E2 -5421.002} C_VEL
LIN {X 0,Y 509.864,Z 218.473,A -85,B 0,C 180,E1 -5424.427,E2 -5424.427} C_VEL
LIN {X 0,Y 509.884,Z 218.464,A -85,B 0,C 180,E1 -5427.056,E2 -5427.056} C_VEL
LIN {X 0,Y 509.857,Z 218.47,A -85,B 0,C 180,E1 -5429.752,E2 -5429.752} C_VEL
LIN {X 0,Y 509.846,Z 218.472,A -85,B 0,C 180,E1 -5432.77,E2 -5432.77} C_VEL
LIN {X 0,Y 509.826,Z 218.472,A -85,B 0,C 180,E1 -5435.579,E2 -5435.579} C_VEL
LIN {X 0,Y 509.851,Z 218.479,A -85,B 0,C 180,E1 -5438.338,E2 -5438.338} C_VEL
LIN {X 0,Y 509.856,Z 218.47,A -85,B 0,C 180,E1 -5441.426,E2 -5441.426} C_VEL
LIN {X 0,Y 509.84,Z 218.476,A -85,B 0,C 180,E1 -5444.67,E2 -5444.67} C_VEL
LIN {X 0,Y 509.835,Z 218.474,A -85,B 0,C 180,E1 -5447.511,E2 -5447.511} C_VEL
LIN {X 0,Y 509.848,Z 218.474,A -85,B 0,C 180,E1 -5450.648,E2 -5450.648} C_VEL
LIN {X 0,Y 509.826,Z 218.477,A -85,B 0,C 180,E1 -5453.647,E2 -5453.647} C_VEL
LIN {X 0,Y 509.861,Z 218.472,A -85,B 0,C 180,E1 -5456.539,E2 -5456.539} C_VEL
LIN {X 0,Y 509.848,Z 218.476,A -85,B 0,C 180,E1 -5459.335,E2 -5459.335} C_VEL
LIN {X 0,Y 509.853,Z 218.476,A -85,B 0,C 180,E1 -5462.052,E2 -5462.052} C_VEL
LIN {X 0,Y 509.95,Z 218.634,A -85,B 0,C 180,E1 -5463.664,E2 -5463.664} C_VEL
LIN {X 0,Y 511.164,Z 226.445,A -85,B 0,C 180,E1 -5465.407,E2 -5465.407} C_VEL
LIN {X 0,Y 510.824,Z 237.871,A -85,B 0,C 180,E1 -5467.769,E2 -5467.769} C_VEL
LIN {X 0,Y 510.544,Z 250.428,A -85,B 0,C 180,E1 -5470.29,E2 -5470.29} C_VEL
LIN {X 0,Y 510.109,Z 265.929,A -85,B 0,C 180,E1 -5473.389,E2 -5473.389} C_VEL
LIN {X 0,Y 509.995,Z 270.994,A -85,B 0,C 180,E1 -5474.391,E2 -5474.391} C_VEL
LIN {X 0,Y 510.752,Z 275.736,A -85,B 0,C 180,E1 -5474.52,E2 -5474.52} C_VEL
LIN {X 0,Y 512.206,Z 285.436,A -85,B 0,C 180,E1 -5474.703,E2 -5474.703} C_VEL
LIN {X 0,Y 511.763,Z 375.944,A -85,B 0,C 180,E1 -5475.993,E2 -5475.993} C_VEL
LIN {X 0,Y 511.586,Z 385.842,A -85,B 0,C 180,E1 -5476.216,E2 -5476.216} C_VEL
LIN {X 0,Y 511.358,Z 395.819,A -85,B 0,C 180,E1 -5476.539,E2 -5476.539} C_VEL
LIN {X 0,Y 511.131,Z 406.186,A -85,B 0,C 180,E1 -5476.988,E2 -5476.988} C_VEL
LIN {X 0,Y 510.855,Z 415.726,A -85,B 0,C 180,E1 -5477.511,E2 -5477.511} C_VEL
LIN {X 0,Y 510.576,Z 424.322,A -85,B 0,C 180,E1 -5478.084,E2 -5478.084} C_VEL
LIN {X 0,Y 510.327,Z 433.054,A -85,B 0,C 180,E1 -5478.783,E2 -5478.783} C_VEL
LIN {X 0,Y 510.044,Z 440.45,A -85,B 0,C 180,E1 -5479.48,E2 -5479.48} C_VEL
LIN {X 0,Y 509.869,Z 447.673,A -85,B 0,C 180,E1 -5480.279,E2 -5480.279} C_VEL
LIN {X 0,Y 509.673,Z 453.875,A -85,B 0,C 180,E1 -5481.076,E2 -5481.076} C_VEL
LIN {X 0,Y 509.504,Z 460.413,A -85,B 0,C 180,E1 -5482.071,E2 -5482.071} C_VEL
LIN {X 0,Y 509.336,Z 465.966,A -85,B 0,C 180,E1 -5483.085,E2 -5483.085} C_VEL
LIN {X 0,Y 509.299,Z 470.403,A -85,B 0,C 180,E1 -5484.06,E2 -5484.06} C_VEL
LIN {X 0,Y 509.191,Z 474.722,A -85,B 0,C 180,E1 -5485.25,E2 -5485.25} C_VEL
LIN {X 0,Y 509.246,Z 477.087,A -85,B 0,C 180,E1 -5486.043,E2 -5486.043} C_VEL
LIN {X 0,Y 509.201,Z 478.882,A -85,B 0,C 180,E1 -5486.835,E2 -5486.835} C_VEL
LIN {X 0,Y 509.113,Z 481.319,A -85,B 0,C 180,E1 -5488.418,E2 -5488.418} C_VEL
LIN {X 0,Y 509.074,Z 481.905,A -85,B 0,C 180,E1 -5489.209,E2 -5489.209} C_VEL
LIN {X 0,Y 509.074,Z 481.905,A -85,B 0,C 180,E1 -5490.791,E2 -5490.791} C_VEL
LIN {X 0,Y 509.113,Z 481.319,A -85,B 0,C 180,E1 -5491.582,E2 -5491.582} C_VEL
LIN {X 0,Y 509.201,Z 478.882,A -85,B 0,C 180,E1 -5493.165,E2 -5493.165} C_VEL
